// TIA Portal project "TronCamTuDong" (V16)

(* hardware
DEVICE "S7-1200 station_1"  S7-1200 Station
   slot 0: "Rack_0"  S7-1200 Rack  Rack  V1.0
   slot 1: "PLC_1"  CPU 1214C AC/DC/Rly  6ES7 214-1BG40-0XB0  V4.2
*)

// ===== PLC "PLC_1"  CPU 1214C AC/DC/Rly =====

VAR_GLOBAL   // PLC tag table "Input"
   "I_Start" AT %I0.0 : Bool;   // Nút nhấn Start
   "I_Stop" AT %I0.1 : Bool;   // Nút nhấn Stop
   "I_Mode" AT %I0.2 : Bool;   // Công tắc chọn chế độ vận hành
   "I_Ss_Low_XiloA1" AT %I0.3 : Bool;   // Cảm biến xi lô A1
   "I_Ss_Low_XiloA2" AT %I0.4 : Bool;   // Cảm biến xi lô A2
   "I_Ss_Low_XiloA3" AT %I0.5 : Bool;   // Cảm biến xi lô A3
   "I_Ss_Low_XiloA4" AT %I0.6 : Bool;   // Cảm biến xi lô A4
   "I_Ss_Low_XiloA5" AT %I0.7 : Bool;   // Cảm biến xi lô A5
   "I_Ss_Low_XiloA6" AT %I1.0 : Bool;   // Cảm biến xi lô A6
   "I_Ss_Low_XiloA7" AT %I1.1 : Bool;   // Cảm biến xi lô A7
   "I_Ss_Low_XiloA8" AT %I1.2 : Bool;   // Cảm biến xi lô A8
   "I_Ss_Low_XiloA9" AT %I1.3 : Bool;   // Cảm biến xi lô A9
   "I_Ss_Low_XiloB1" AT %I1.4 : Bool;   // Cảm biến xi lô B1
   "I_Ss_Low_XiloB2" AT %I1.5 : Bool;   // Cảm biến xi lô B2
   "I_Ss_Low_XiloB3" AT %I1.6 : Bool;   // Cảm biến xi lô B3
   "I_Ss_Low_XiloB4" AT %I1.7 : Bool;   // Cảm biến xi lô B4
   "I_Ss_Low_XiloB5" AT %I2.0 : Bool;   // Cảm biến xi lô B5
   "I_Ss_Low_XiloB6" AT %I2.1 : Bool;   // Cảm biến xi lô B6
   "I_Ss_Low_XiloB7" AT %I2.2 : Bool;   // Cảm biến xi lô B7
   "I_Ss_ValvesA" AT %I2.3 : Bool;   // Cảm biến van ở thùng cân A
   "I_Ss_ValvesB" AT %I2.4 : Bool;   // Cảm biến van ở thùng cân B
   "I_Ss_Tank_Low" AT %I2.5 : Bool;   // Cảm biến mức thấp bình trộn
   "I_Ss_Tank_High" AT %I2.6 : Bool;   // Cảm biến mức cao bình trộn
   "I_Ss_Valves_Out" AT %I2.7 : Bool;   // Cảm biến van xả ở bình trộn
   "I_SW_Motor_Tai" AT %I3.0 : Bool;   // Công tắc chế độ thủ công động cơ vít tải
   "I_SW_Motor_Mixed" AT %I3.1 : Bool;   // Công tắc chế độ thủ công động cơ trộn
   "I_SW_ValvesA" AT %I3.2 : Bool;   // Công tắc chế độ thủ công van xả thùng cân A
   "I_SW_ValvesB" AT %I3.3 : Bool;   // Công tắc chế độ thủ công van xả thùng cân B
   "I_SW_Valves_Out" AT %I3.4 : Bool;   // Công tắc chế độ thủ công van xả bình trộn
   "I_Load_ScalesA" AT %ID4 : Real;   // Cảm biến cân thùng cân A
   "I_Load_ScalesB" AT %ID8 : Real;   // Cảm biến cân thùng cân B
END_VAR

VAR_GLOBAL   // PLC tag table "Output"
   "Q_lamp_Auto" AT %Q0.0 : Bool;   // Đèn báo chế độ tự động
   "Q_lamp_Manu" AT %Q0.1 : Bool;   // Đèn báo chế độ thủ công
   "Q_lamp_Fault" AT %Q0.2 : Bool;   // Đèn báo lỗi
   "Q_Motor_Tai" AT %Q0.3 : Bool;   // Động cơ vít tải
   "Q_ValveA" AT %Q0.4 : Bool;   // Van xả thùng cân A
   "Q_ValveB" AT %Q0.5 : Bool;   // Van xả thùng cân B
   "Q_Valve_Out" AT %Q0.6 : Bool;   // Van xả bình trộn
   "Q_Motor_Mixed" AT %Q0.7 : Bool;   // Động cơ trộn
   "Q_Motor_Conveyor" AT %Q1.0 : Bool;   // Động cơ điều khiển băng tải
END_VAR

VAR_GLOBAL   // PLC tag table "Output_Auto"
   "M_Auto_Motor_Tai" AT %M20.0 : Bool;
   "M_Auto_ValveA" AT %M20.1 : Bool;
   "M_Auto_ValveB" AT %M20.2 : Bool;
   "M_Auto_Valve_Out" AT %M20.3 : Bool;
   "M_Auto_Motor_Mixed" AT %M20.4 : Bool;
END_VAR

VAR_GLOBAL   // PLC tag table "Output_Manu"
   "M_Manu_Motor_Tai" AT %M30.0 : Bool;
   "M_Manu_ValveA" AT %M30.1 : Bool;
   "M_Manu_ValveB" AT %M30.2 : Bool;
   "M_Manu_Valve_Out" AT %M30.3 : Bool;
   "M_Manu_Motor_Mixed" AT %M30.4 : Bool;
END_VAR

VAR_GLOBAL   // PLC tag table "TrungGian"
   "M_LoadXilo" AT %M15.0 : Bool;
   "M_DK_VanHanh" AT %M15.1 : Bool;
   "M_Step1" AT %M15.2 : Bool;
   "M_Step3" AT %M15.4 : Bool;
   "M_Xung200ms" AT %M15.5 : Bool;
   "M_TG_Laplai" AT %M16.3 : Bool;
   "M_CloseValve1" AT %M16.4 : Bool;
   "M_CloseValve2" AT %M16.5 : Bool;
   "M_Close_MotorTai" AT %M16.6 : Bool;
   "M_Close_MotorMixed" AT %M16.7 : Bool;
   "M_Close_ValveOut" AT %M17.0 : Bool;
   "M_Reset" AT %M17.1 : Bool;
   "M_Step2" AT %M15.3 : Bool;
END_VAR

VAR_GLOBAL   // PLC tag table "TG_Cell_Xilo"
   "M_ScalesA" AT %MD120 : Real;
   "M_ScalesB" AT %MD124 : Real;
   "M_Inverter" AT %MD148 : Real;
END_VAR

DATA_BLOCK "Input"   // DB1
{ S7_Optimized_Access := 'FALSE' }
VERSION : 0.1
   VAR
      Start : Bool;
      Stop : Bool;
      Mode : Bool;
      Simulation : Bool;
      Ss_Low_XiloA1 : Bool;
      Ss_Low_XiloA2 : Bool;
      Ss_Low_XiloA3 : Bool;
      Ss_Low_XiloA4 : Bool;
      Ss_Low_XiloA5 : Bool;
      Ss_Low_XiloA6 : Bool;
      Ss_Low_XiloA7 : Bool;
      Ss_Low_XiloA8 : Bool;
      Ss_Low_XiloA9 : Bool;
      Ss_Low_XiloB1 : Bool;
      Ss_Low_XiloB2 : Bool;
      Ss_Low_XiloB3 : Bool;
      Ss_Low_XiloB4 : Bool;
      Ss_Low_XiloB5 : Bool;
      Ss_Low_XiloB6 : Bool;
      Ss_Low_XiloB7 : Bool;
      Ss_ScalesA : Bool;
      Ss_ScalesB : Bool;
      Ss_Tank_Low : Bool;
      Ss_Tank_High : Bool;
      Ss_Valves_Out : Bool;
      SW_Motor_Tai : Bool;
      SW_Motor_Mixed : Bool;
      SW_ValvesA : Bool;
      SW_ValvesB : Bool;
      SW_Valves_Out : Bool;
   END_VAR
BEGIN
END_DATA_BLOCK

DATA_BLOCK "Output"   // DB2
{ S7_Optimized_Access := 'FALSE' }
VERSION : 0.1
   VAR
      Lamp_Auto : Bool;
      Lamp_Manu : Bool;
      Lamp_Fault : Bool;
      Motor_Tai : Bool;
      ValveA : Bool;
      ValveB : Bool;
      Valve_Out : Bool;
      Motor_Mixed : Bool;
      EndSystem : Bool;
      Act_SoMeTron : Int;
      Act_Weight_XiloA1 : Real;
      Act_Weight_XiloA2 : Real;
      Act_Weight_XiloA3 : Real;
      Act_Weight_XiloA4 : Real;
      Act_Weight_XiloA5 : Real;
      Act_Weight_XiloA6 : Real;
      Act_Weight_XiloA7 : Real;
      Act_Weight_XiloA8 : Real;
      Act_Weight_XiloA9 : Real;
      Act_Weight_XiloB1 : Real;
      Act_Weight_XiloB2 : Real;
      Act_Weight_XiloB3 : Real;
      Act_Weight_XiloB4 : Real;
      Act_Weight_XiloB5 : Real;
      Act_Weight_XiloB6 : Real;
      Act_Weight_XiloB7 : Real;
      Act_Time_Xa : DInt;
      Act_Time_Tron : DInt;
   END_VAR
BEGIN
END_DATA_BLOCK

DATA_BLOCK "Input_Data"   // DB10
{ S7_Optimized_Access := 'FALSE' }
VERSION : 0.1
   VAR
      Load_ScaleA : Real;
      Load_ScaleB : Real;
      Set_Weight_Gao : Real;
      Set_Weight_Ngo : Real;
      Set_Weight_San : Real;
      Set_Weight_DauKho : Real;
      Set_Weight_BotCa : Real;
      Set_Time_Xa : DInt;
      Set_Time_Tron : DInt;
      Set_SoMeTron : Int;
   END_VAR
BEGIN
END_DATA_BLOCK

DATA_BLOCK "DB_TrungGian"   // DB11
{ S7_Optimized_Access := 'FALSE' }
VERSION : 0.1
   VAR
      Enable_XiloGao : Bool;
      Enable_XiloNgo : Bool;
      Enable_XiloSan : Bool;
      Enable_XiloDauKho : Bool;
      Enable_XiloBotca : Bool;
      Xung_200ms : Bool;
   END_VAR
BEGIN
END_DATA_BLOCK

// folder: System blocks/Program resources

DATA_BLOCK "Xung200ms"   // DB3
{ S7_Optimized_Access := 'TRUE' }
AUTHOR : Simatic
FAMILY : IEC
NAME : IEC_TMR
VERSION : 1.0
// stored: InstanceOfName IEC_TIMER
"IEC_TIMER"
BEGIN
END_DATA_BLOCK

DATA_BLOCK "Time_Mix"   // DB4
{ S7_Optimized_Access := 'TRUE' }
AUTHOR : Simatic
FAMILY : IEC
NAME : IEC_TMR
VERSION : 1.0
// stored: InstanceOfName IEC_TIMER
"IEC_TIMER"
BEGIN
END_DATA_BLOCK

DATA_BLOCK "Time_Xa"   // DB5
{ S7_Optimized_Access := 'TRUE' }
AUTHOR : Simatic
FAMILY : IEC
NAME : IEC_TMR
VERSION : 1.0
// stored: InstanceOfName IEC_TIMER
"IEC_TIMER"
BEGIN
END_DATA_BLOCK

DATA_BLOCK "TimeDelay"   // DB6
{ S7_Optimized_Access := 'TRUE' }
AUTHOR : Simatic
FAMILY : IEC
NAME : IEC_TMR
VERSION : 1.0
// stored: InstanceOfName IEC_TIMER
"IEC_TIMER"
BEGIN
END_DATA_BLOCK

DATA_BLOCK "TimeDelay2"   // DB7
{ S7_Optimized_Access := 'TRUE' }
AUTHOR : Simatic
FAMILY : IEC
NAME : IEC_TMR
VERSION : 1.0
// stored: InstanceOfName IEC_TIMER
"IEC_TIMER"
BEGIN
END_DATA_BLOCK

DATA_BLOCK "Dem_SoMe"   // DB8
{ S7_Optimized_Access := 'TRUE' }
AUTHOR : Simatic
FAMILY : IEC
NAME : CNTR
VERSION : 1.0
// stored: InstanceOfName IEC_COUNTER
"IEC_COUNTER"
BEGIN
END_DATA_BLOCK

DATA_BLOCK "Time_Delay3"   // DB9
{ S7_Optimized_Access := 'TRUE' }
AUTHOR : Simatic
FAMILY : IEC
NAME : IEC_TMR
VERSION : 1.0
// stored: InstanceOfName IEC_TIMER
"IEC_TIMER"
BEGIN
END_DATA_BLOCK

// folder: (top level)

FUNCTION "FC_Auto" : Void   // FC1, LAD
{ S7_Optimized_Access := 'TRUE' }
VERSION : 0.1
   VAR_TEMP   // added for the SCL form of the ladder/FBD networks
      _w1 : Bool;
   END_VAR
BEGIN

REGION Network 1: kiểm tra điều kiện các giá trị khối lượng n.liệu và t.gian xả , trộn > 0
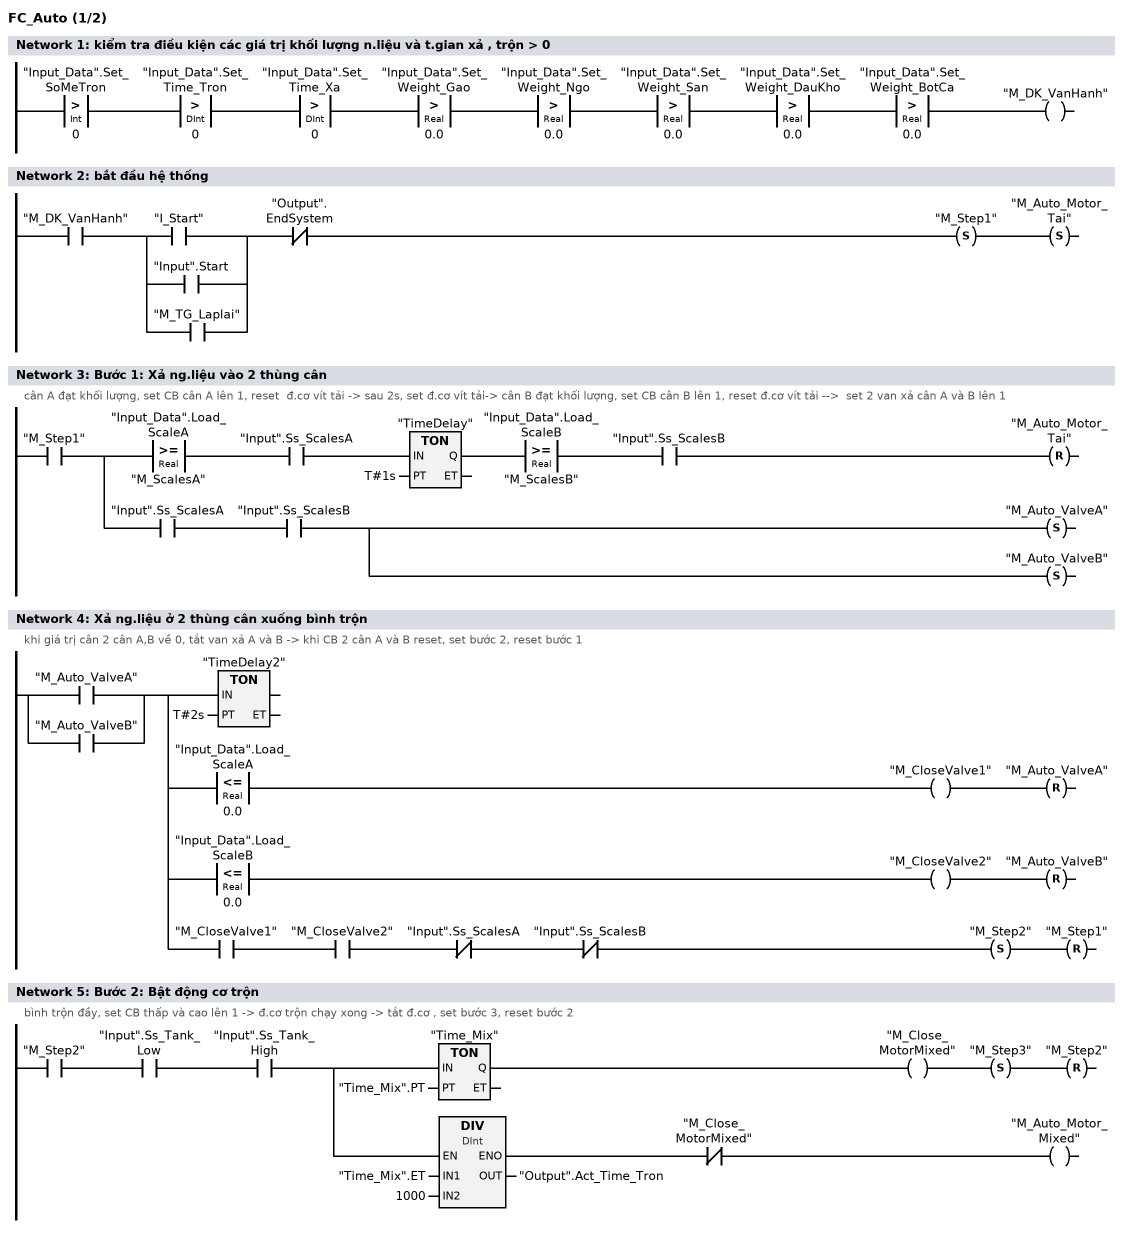
   RUNG wire#powerrail
      { S7_Templates := "SrcType := Int" } GT_Contact(in1 := "Input_Data".Set_SoMeTron, in2 := 0)
      { S7_Templates := "SrcType := DInt" } GT_Contact(in1 := "Input_Data".Set_Time_Tron, in2 := 0)
      { S7_Templates := "SrcType := DInt" } GT_Contact(in1 := "Input_Data".Set_Time_Xa, in2 := 0)
      { S7_Templates := "SrcType := Real" } GT_Contact(in1 := "Input_Data".Set_Weight_Gao, in2 := 0.0)
      { S7_Templates := "SrcType := Real" } GT_Contact(in1 := "Input_Data".Set_Weight_Ngo, in2 := 0.0)
      { S7_Templates := "SrcType := Real" } GT_Contact(in1 := "Input_Data".Set_Weight_San, in2 := 0.0)
      { S7_Templates := "SrcType := Real" } GT_Contact(in1 := "Input_Data".Set_Weight_DauKho, in2 := 0.0)
      { S7_Templates := "SrcType := Real" } GT_Contact(in1 := "Input_Data".Set_Weight_BotCa, in2 := 0.0)
      Coil( "M_DK_VanHanh" )
   END_RUNG
   // the same network as SCL:
   "M_DK_VanHanh" := ("Input_Data".Set_SoMeTron > 0) AND ("Input_Data".Set_Time_Tron > 0) AND ("Input_Data".Set_Time_Xa > 0) AND ("Input_Data".Set_Weight_Gao > 0.0) AND ("Input_Data".Set_Weight_Ngo > 0.0) AND ("Input_Data".Set_Weight_San > 0.0) AND ("Input_Data".Set_Weight_DauKho > 0.0) AND ("Input_Data".Set_Weight_BotCa > 0.0);
END_REGION

REGION Network 2: bắt đầu hệ thống
   RUNG wire#powerrail
      Contact( "M_DK_VanHanh" )
      wire#w1
      Contact( "I_Start" )
      wire#w2
      I_Contact( "Output".EndSystem )
      S_Coil( "M_Step1" )
      S_Coil( "M_Auto_Motor_Tai" )
   END_RUNG
   RUNG wire#w1
      Contact( "Input".Start )
   END_RUNG wire#w2
   RUNG wire#w1
      Contact( "M_TG_Laplai" )
   END_RUNG wire#w2
   // the same network as SCL:
   IF "M_DK_VanHanh" AND ("I_Start" OR "Input".Start OR "M_TG_Laplai") AND NOT "Output".EndSystem THEN
       "M_Step1" := TRUE;
       "M_Auto_Motor_Tai" := TRUE;
   END_IF;
END_REGION

REGION Network 3: Bước 1: Xả ng.liệu vào 2 thùng cân
   // cân A đạt khối lượng, set CB cân A lên 1, reset  đ.cơ vít tải -> sau 2s, set đ.cơ vít tải-> cân B đạt khối lượng, set CB cân B lên 1, reset đ.cơ vít tải -->  set 2 van xả cân A và B lên 1
   "TimeDelay".TON(IN := "M_Step1" AND ("Input_Data".Load_ScaleA >= "M_ScalesA") AND "Input".Ss_ScalesA,
                   PT := T#1s);
   IF "TimeDelay".Q AND ("Input_Data".Load_ScaleB >= "M_ScalesB") AND "Input".Ss_ScalesB THEN
       "M_Auto_Motor_Tai" := FALSE;
   END_IF;
   IF "M_Step1" AND "Input".Ss_ScalesA AND "Input".Ss_ScalesB THEN
       "M_Auto_ValveA" := TRUE;
       "M_Auto_ValveB" := TRUE;
   END_IF;
END_REGION

REGION Network 4: Xả ng.liệu ở 2 thùng cân xuống bình trộn
   // khi giá trị cân 2 cân A,B về 0, tắt van xả A và B -> khi CB 2 cân A và B reset, set bước 2, reset bước 1
   #_w1 := "M_Auto_ValveA" OR "M_Auto_ValveB";
   "TimeDelay2".TON(IN := #_w1, PT := T#2s);
   "M_CloseValve1" := #_w1 AND ("Input_Data".Load_ScaleA <= 0.0);
   IF "M_CloseValve1" THEN "M_Auto_ValveA" := FALSE; END_IF;
   "M_CloseValve2" := #_w1 AND ("Input_Data".Load_ScaleB <= 0.0);
   IF "M_CloseValve2" THEN "M_Auto_ValveB" := FALSE; END_IF;
   IF #_w1 AND "M_CloseValve1" AND "M_CloseValve2" AND NOT "Input".Ss_ScalesA AND NOT "Input".Ss_ScalesB THEN
       "M_Step2" := TRUE;
       "M_Step1" := FALSE;
   END_IF;
END_REGION

REGION Network 5: Bước 2: Bật động cơ trộn
   // bình trộn đầy, set CB thấp và cao lên 1 -> đ.cơ trộn chạy xong -> tắt đ.cơ , set bước 3, reset bước 2
   #_w1 := "M_Step2" AND "Input".Ss_Tank_Low AND "Input".Ss_Tank_High;
   "Time_Mix".TON(IN := #_w1, PT := "Time_Mix".PT);
   "M_Close_MotorMixed" := "Time_Mix".Q;
   IF "Time_Mix".Q THEN
       "M_Step3" := TRUE;
       "M_Step2" := FALSE;
   END_IF;
   IF #_w1 THEN "Output".Act_Time_Tron := "Time_Mix".ET / 1000; END_IF;
   "M_Auto_Motor_Mixed" := #_w1 AND NOT "M_Close_MotorMixed";
END_REGION

REGION Network 6: Bước 3: bật van xả liệu đầu ra
   // CB cao bình trộn reset , bắt đầu xả -> xả xong , CB thấp reset , tắt van xả đầu ra --> set biến lặp lại, reset bước 3
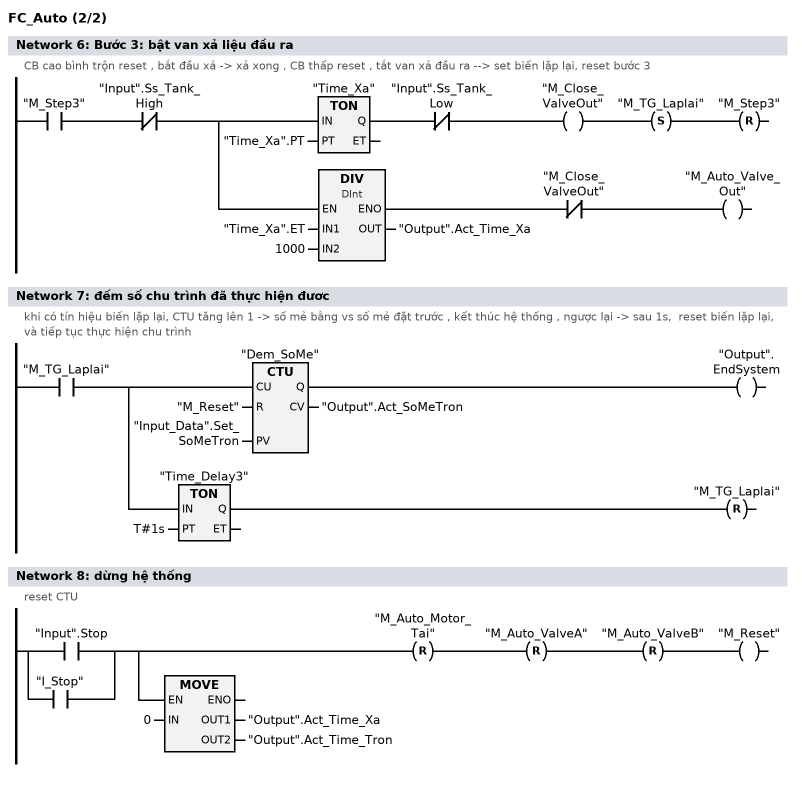
   #_w1 := "M_Step3" AND NOT "Input".Ss_Tank_High;
   "Time_Xa".TON(IN := #_w1, PT := "Time_Xa".PT);
   "M_Close_ValveOut" := "Time_Xa".Q AND NOT "Input".Ss_Tank_Low;
   IF "M_Close_ValveOut" THEN
       "M_TG_Laplai" := TRUE;
       "M_Step3" := FALSE;
   END_IF;
   IF #_w1 THEN "Output".Act_Time_Xa := "Time_Xa".ET / 1000; END_IF;
   "M_Auto_Valve_Out" := #_w1 AND NOT "M_Close_ValveOut";
END_REGION

REGION Network 7: đếm số chu trình đã thực hiện đươc
   // khi có tín hiệu biến lặp lại, CTU tăng lên 1 -> số mẻ bằng vs số mẻ đặt trước , kết thúc hệ thống , ngược lại -> sau 1s,  reset biến lặp lại, và tiếp tục thực hiện chu trình
   "Dem_SoMe".CTU(CU := "M_TG_Laplai",
                  R := "M_Reset",
                  PV := "Input_Data".Set_SoMeTron,
                  CV => "Output".Act_SoMeTron);
   "Output".EndSystem := "Dem_SoMe".Q;
   "Time_Delay3".TON(IN := "M_TG_Laplai", PT := T#1s);
   IF "Time_Delay3".Q THEN "M_TG_Laplai" := FALSE; END_IF;
END_REGION

REGION Network 8: dừng hệ thống
   // reset CTU
   RUNG wire#powerrail
      Contact( "Input".Stop )
      wire#w1
      R_Coil( "M_Auto_Motor_Tai" )
      R_Coil( "M_Auto_ValveA" )
      R_Coil( "M_Auto_ValveB" )
      Coil( "M_Reset" )
   END_RUNG
   RUNG wire#powerrail
      Contact( "I_Stop" )
   END_RUNG wire#w1
   RUNG wire#w1
      Move(in := 0, out1 => "Output".Act_Time_Xa, out2 => "Output".Act_Time_Tron)
   END_RUNG
   // the same network as SCL:
   #_w1 := "Input".Stop OR "I_Stop";
   IF #_w1 THEN
       "M_Auto_Motor_Tai" := FALSE;
       "M_Auto_ValveA" := FALSE;
       "M_Auto_ValveB" := FALSE;
   END_IF;
   "M_Reset" := #_w1;
   IF #_w1 THEN
       "Output".Act_Time_Xa := 0;
       "Output".Act_Time_Tron := 0;
   END_IF;
END_REGION
END_FUNCTION

FUNCTION "FC_Manu" : Void   // FC2, LAD
{ S7_Optimized_Access := 'TRUE' }
VERSION : 0.1
BEGIN

REGION Network 1: bật/ tắt đ.cơ tải
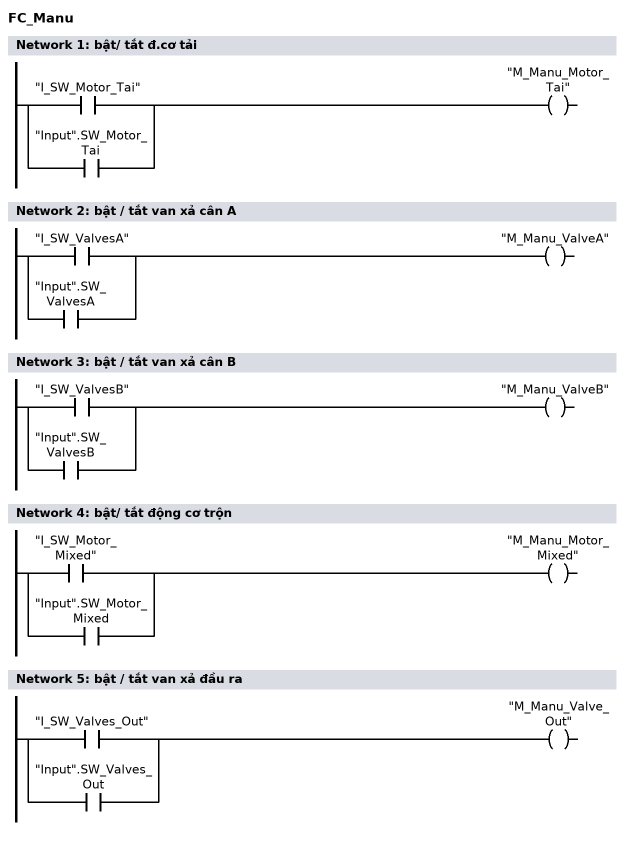
   RUNG wire#powerrail
      Contact( "I_SW_Motor_Tai" )
      wire#w1
      Coil( "M_Manu_Motor_Tai" )
   END_RUNG
   RUNG wire#powerrail
      Contact( "Input".SW_Motor_Tai )
   END_RUNG wire#w1
   // the same network as SCL:
   "M_Manu_Motor_Tai" := "I_SW_Motor_Tai" OR "Input".SW_Motor_Tai;
END_REGION

REGION Network 2: bật / tắt van xả cân A
   RUNG wire#powerrail
      Contact( "I_SW_ValvesA" )
      wire#w1
      Coil( "M_Manu_ValveA" )
   END_RUNG
   RUNG wire#powerrail
      Contact( "Input".SW_ValvesA )
   END_RUNG wire#w1
   // the same network as SCL:
   "M_Manu_ValveA" := "I_SW_ValvesA" OR "Input".SW_ValvesA;
END_REGION

REGION Network 3: bật / tắt van xả cân B
   RUNG wire#powerrail
      Contact( "I_SW_ValvesB" )
      wire#w1
      Coil( "M_Manu_ValveB" )
   END_RUNG
   RUNG wire#powerrail
      Contact( "Input".SW_ValvesB )
   END_RUNG wire#w1
   // the same network as SCL:
   "M_Manu_ValveB" := "I_SW_ValvesB" OR "Input".SW_ValvesB;
END_REGION

REGION Network 4: bật/ tắt động cơ trộn
   RUNG wire#powerrail
      Contact( "I_SW_Motor_Mixed" )
      wire#w1
      Coil( "M_Manu_Motor_Mixed" )
   END_RUNG
   RUNG wire#powerrail
      Contact( "Input".SW_Motor_Mixed )
   END_RUNG wire#w1
   // the same network as SCL:
   "M_Manu_Motor_Mixed" := "I_SW_Motor_Mixed" OR "Input".SW_Motor_Mixed;
END_REGION

REGION Network 5: bật / tắt van xả đầu ra
   RUNG wire#powerrail
      Contact( "I_SW_Valves_Out" )
      wire#w1
      Coil( "M_Manu_Valve_Out" )
   END_RUNG
   RUNG wire#powerrail
      Contact( "Input".SW_Valves_Out )
   END_RUNG wire#w1
   // the same network as SCL:
   "M_Manu_Valve_Out" := "I_SW_Valves_Out" OR "Input".SW_Valves_Out;
END_REGION
END_FUNCTION

FUNCTION "FC_Simulation" : Void   // FC3, LAD
{ S7_Optimized_Access := 'TRUE' }
VERSION : 0.1
   VAR_TEMP   // added for the SCL form of the ladder/FBD networks
      _w1 : Bool;
      _w2 : Bool;
      _w3 : Bool;
      _w4 : Bool;
   END_VAR
BEGIN

REGION Network 1: tạo xung 200ms
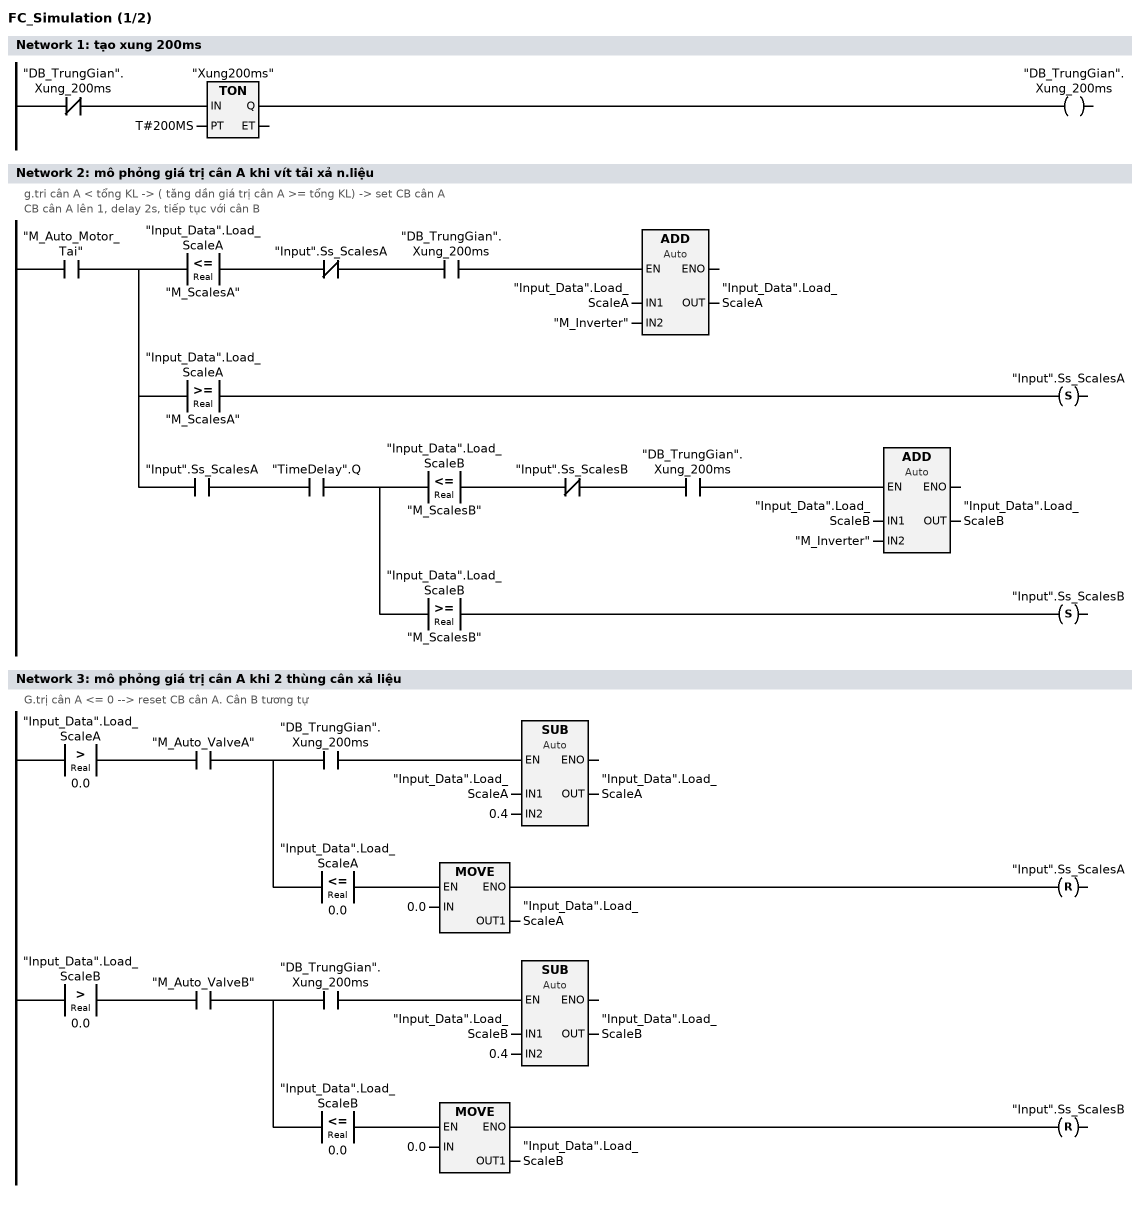
   "Xung200ms".TON(IN := NOT "DB_TrungGian".Xung_200ms, PT := T#200MS);
   "DB_TrungGian".Xung_200ms := "Xung200ms".Q;
END_REGION

REGION Network 2: mô phỏng giá trị cân A khi vít tải xả n.liệu
   // g.tri cân A < tổng KL -> ( tăng dần giá trị cân A >= tổng KL) -> set CB cân A 
   // CB cân A lên 1, delay 2s, tiếp tục với cân B
   RUNG wire#powerrail
      Contact( "M_Auto_Motor_Tai" )
      wire#w1
      { S7_Templates := "SrcType := Real" } LE_Contact(in1 := "Input_Data".Load_ScaleA, in2 := "M_ScalesA")
      I_Contact( "Input".Ss_ScalesA )
      Contact( "DB_TrungGian".Xung_200ms )
      Add(in1 := "Input_Data".Load_ScaleA, in2 := "M_Inverter", out => "Input_Data".Load_ScaleA)
   END_RUNG
   RUNG wire#w1
      { S7_Templates := "SrcType := Real" } GE_Contact(in1 := "Input_Data".Load_ScaleA, in2 := "M_ScalesA")
      S_Coil( "Input".Ss_ScalesA )
   END_RUNG
   RUNG wire#w1
      Contact( "Input".Ss_ScalesA )
      Contact( "TimeDelay".Q )
      wire#w2
      { S7_Templates := "SrcType := Real" } LE_Contact(in1 := "Input_Data".Load_ScaleB, in2 := "M_ScalesB")
      I_Contact( "Input".Ss_ScalesB )
      Contact( "DB_TrungGian".Xung_200ms )
      Add(in1 := "Input_Data".Load_ScaleB, in2 := "M_Inverter", out => "Input_Data".Load_ScaleB)
   END_RUNG
   RUNG wire#w2
      { S7_Templates := "SrcType := Real" } GE_Contact(in1 := "Input_Data".Load_ScaleB, in2 := "M_ScalesB")
      S_Coil( "Input".Ss_ScalesB )
   END_RUNG
   // the same network as SCL:
   IF "M_Auto_Motor_Tai" AND ("Input_Data".Load_ScaleA <= "M_ScalesA") AND NOT "Input".Ss_ScalesA AND "DB_TrungGian".Xung_200ms THEN
       "Input_Data".Load_ScaleA := "Input_Data".Load_ScaleA + "M_Inverter";
   END_IF;
   IF "M_Auto_Motor_Tai" AND ("Input_Data".Load_ScaleA >= "M_ScalesA") THEN
       "Input".Ss_ScalesA := TRUE;
   END_IF;
   #_w1 := "M_Auto_Motor_Tai" AND "Input".Ss_ScalesA AND "TimeDelay".Q;
   IF #_w1 AND ("Input_Data".Load_ScaleB <= "M_ScalesB") AND NOT "Input".Ss_ScalesB AND "DB_TrungGian".Xung_200ms THEN
       "Input_Data".Load_ScaleB := "Input_Data".Load_ScaleB + "M_Inverter";
   END_IF;
   IF #_w1 AND ("Input_Data".Load_ScaleB >= "M_ScalesB") THEN "Input".Ss_ScalesB := TRUE; END_IF;
END_REGION

REGION Network 3: mô phỏng giá trị cân A khi 2 thùng cân xả liệu
   // G.trị cân A <= 0 --> reset CB cân A. Cân B tương tự
   RUNG wire#powerrail
      { S7_Templates := "SrcType := Real" } GT_Contact(in1 := "Input_Data".Load_ScaleA, in2 := 0.0)
      Contact( "M_Auto_ValveA" )
      wire#w1
      Contact( "DB_TrungGian".Xung_200ms )
      Sub(in1 := "Input_Data".Load_ScaleA, in2 := 0.4, out => "Input_Data".Load_ScaleA)
   END_RUNG
   RUNG wire#w1
      { S7_Templates := "SrcType := Real" } LE_Contact(in1 := "Input_Data".Load_ScaleA, in2 := 0.0)
      Move(in := 0.0, out1 => "Input_Data".Load_ScaleA)
      R_Coil( "Input".Ss_ScalesA )
   END_RUNG
   RUNG wire#powerrail
      { S7_Templates := "SrcType := Real" } GT_Contact(in1 := "Input_Data".Load_ScaleB, in2 := 0.0)
      Contact( "M_Auto_ValveB" )
      wire#w2
      Contact( "DB_TrungGian".Xung_200ms )
      Sub(in1 := "Input_Data".Load_ScaleB, in2 := 0.4, out => "Input_Data".Load_ScaleB)
   END_RUNG
   RUNG wire#w2
      { S7_Templates := "SrcType := Real" } LE_Contact(in1 := "Input_Data".Load_ScaleB, in2 := 0.0)
      Move(in := 0.0, out1 => "Input_Data".Load_ScaleB)
      R_Coil( "Input".Ss_ScalesB )
   END_RUNG
   // the same network as SCL:
   #_w1 := ("Input_Data".Load_ScaleA > 0.0) AND "M_Auto_ValveA";
   IF #_w1 AND "DB_TrungGian".Xung_200ms THEN
       "Input_Data".Load_ScaleA := "Input_Data".Load_ScaleA - 0.4;
   END_IF;
   #_w2 := #_w1 AND ("Input_Data".Load_ScaleA <= 0.0);
   IF #_w2 THEN
       "Input_Data".Load_ScaleA := 0.0;
       "Input".Ss_ScalesA := FALSE;
   END_IF;
   #_w3 := ("Input_Data".Load_ScaleB > 0.0) AND "M_Auto_ValveB";
   IF #_w3 AND "DB_TrungGian".Xung_200ms THEN
       "Input_Data".Load_ScaleB := "Input_Data".Load_ScaleB - 0.4;
   END_IF;
   #_w4 := #_w3 AND ("Input_Data".Load_ScaleB <= 0.0);
   IF #_w4 THEN
       "Input_Data".Load_ScaleB := 0.0;
       "Input".Ss_ScalesB := FALSE;
   END_IF;
END_REGION

REGION Network 4
   // Khi 2 thùng cân bắt đầu xả , sau 2s , set CB thấp. Sau khi xả hết 2 thùng, set bước 2 và set CB cao
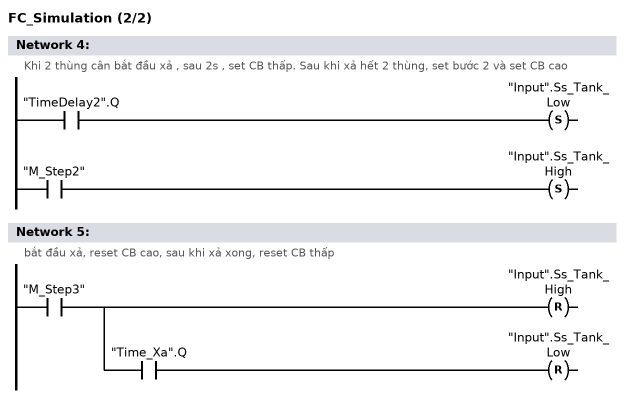
   RUNG wire#powerrail
      Contact( "TimeDelay2".Q )
      S_Coil( "Input".Ss_Tank_Low )
   END_RUNG
   RUNG wire#powerrail
      Contact( "M_Step2" )
      S_Coil( "Input".Ss_Tank_High )
   END_RUNG
   // the same network as SCL:
   IF "TimeDelay2".Q THEN "Input".Ss_Tank_Low := TRUE; END_IF;
   IF "M_Step2" THEN "Input".Ss_Tank_High := TRUE; END_IF;
END_REGION

REGION Network 5
   // bắt đầu xả, reset CB cao, sau khi xả xong, reset CB thấp
   RUNG wire#powerrail
      Contact( "M_Step3" )
      wire#w1
      R_Coil( "Input".Ss_Tank_High )
   END_RUNG
   RUNG wire#w1
      Contact( "Time_Xa".Q )
      R_Coil( "Input".Ss_Tank_Low )
   END_RUNG
   // the same network as SCL:
   IF "M_Step3" THEN "Input".Ss_Tank_High := FALSE; END_IF;
   IF "M_Step3" AND "Time_Xa".Q THEN "Input".Ss_Tank_Low := FALSE; END_IF;
END_REGION
END_FUNCTION

FUNCTION "FC_Output" : Void   // FC4, LAD
{ S7_Optimized_Access := 'TRUE' }
VERSION : 0.1
// set tín hiệu ngõ ra nếu có tín hiệu từ output manu hoặc auto, ngược lại reset tin hiệu
BEGIN

REGION Network 1
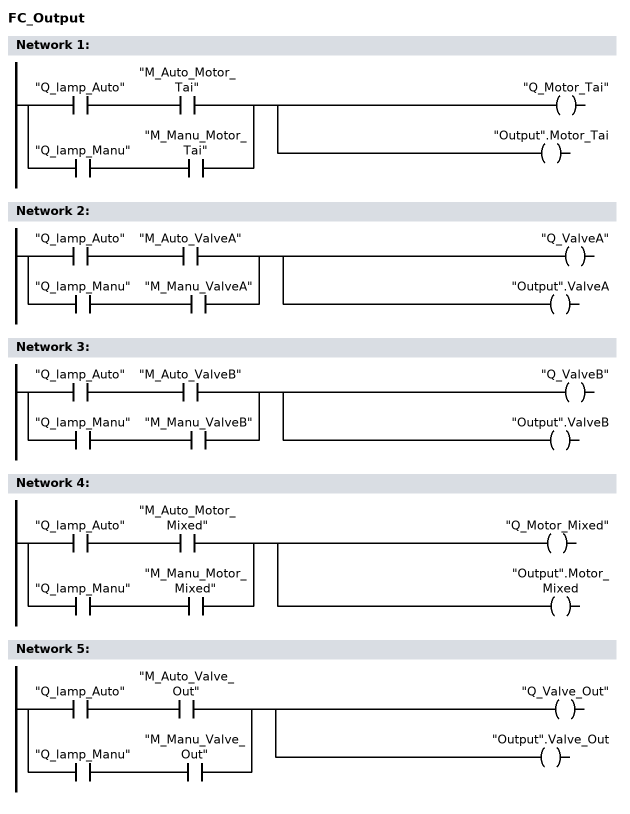
   RUNG wire#powerrail
      Contact( "Q_lamp_Auto" )
      Contact( "M_Auto_Motor_Tai" )
      wire#w1
      Coil( "Q_Motor_Tai" )
   END_RUNG
   RUNG wire#powerrail
      Contact( "Q_lamp_Manu" )
      Contact( "M_Manu_Motor_Tai" )
   END_RUNG wire#w1
   RUNG wire#w1
      Coil( "Output".Motor_Tai )
   END_RUNG
   // the same network as SCL:
   "Q_Motor_Tai" := ("Q_lamp_Auto" AND "M_Auto_Motor_Tai") OR ("Q_lamp_Manu" AND "M_Manu_Motor_Tai");
   "Output".Motor_Tai := "Q_Motor_Tai";
END_REGION

REGION Network 2
   RUNG wire#powerrail
      Contact( "Q_lamp_Auto" )
      Contact( "M_Auto_ValveA" )
      wire#w1
      Coil( "Q_ValveA" )
   END_RUNG
   RUNG wire#powerrail
      Contact( "Q_lamp_Manu" )
      Contact( "M_Manu_ValveA" )
   END_RUNG wire#w1
   RUNG wire#w1
      Coil( "Output".ValveA )
   END_RUNG
   // the same network as SCL:
   "Q_ValveA" := ("Q_lamp_Auto" AND "M_Auto_ValveA") OR ("Q_lamp_Manu" AND "M_Manu_ValveA");
   "Output".ValveA := "Q_ValveA";
END_REGION

REGION Network 3
   RUNG wire#powerrail
      Contact( "Q_lamp_Auto" )
      Contact( "M_Auto_ValveB" )
      wire#w1
      Coil( "Q_ValveB" )
   END_RUNG
   RUNG wire#powerrail
      Contact( "Q_lamp_Manu" )
      Contact( "M_Manu_ValveB" )
   END_RUNG wire#w1
   RUNG wire#w1
      Coil( "Output".ValveB )
   END_RUNG
   // the same network as SCL:
   "Q_ValveB" := ("Q_lamp_Auto" AND "M_Auto_ValveB") OR ("Q_lamp_Manu" AND "M_Manu_ValveB");
   "Output".ValveB := "Q_ValveB";
END_REGION

REGION Network 4
   RUNG wire#powerrail
      Contact( "Q_lamp_Auto" )
      Contact( "M_Auto_Motor_Mixed" )
      wire#w1
      Coil( "Q_Motor_Mixed" )
   END_RUNG
   RUNG wire#powerrail
      Contact( "Q_lamp_Manu" )
      Contact( "M_Manu_Motor_Mixed" )
   END_RUNG wire#w1
   RUNG wire#w1
      Coil( "Output".Motor_Mixed )
   END_RUNG
   // the same network as SCL:
   "Q_Motor_Mixed" := ("Q_lamp_Auto" AND "M_Auto_Motor_Mixed") OR ("Q_lamp_Manu" AND "M_Manu_Motor_Mixed");
   "Output".Motor_Mixed := "Q_Motor_Mixed";
END_REGION

REGION Network 5
   RUNG wire#powerrail
      Contact( "Q_lamp_Auto" )
      Contact( "M_Auto_Valve_Out" )
      wire#w1
      Coil( "Q_Valve_Out" )
   END_RUNG
   RUNG wire#powerrail
      Contact( "Q_lamp_Manu" )
      Contact( "M_Manu_Valve_Out" )
   END_RUNG wire#w1
   RUNG wire#w1
      Coil( "Output".Valve_Out )
   END_RUNG
   // the same network as SCL:
   "Q_Valve_Out" := ("Q_lamp_Auto" AND "M_Auto_Valve_Out") OR ("Q_lamp_Manu" AND "M_Manu_Valve_Out");
   "Output".Valve_Out := "Q_Valve_Out";
END_REGION
END_FUNCTION

FUNCTION "FC_Math" : Void   // FC5, LAD
{ S7_Optimized_Access := 'TRUE' }
VERSION : 0.1
   VAR_TEMP
      sumGaoNgo : Real;
      sumGaoSan : Real;
      sumNgoSan : Real;
   END_VAR
   VAR_TEMP   // added for the SCL form of the ladder/FBD networks
      _w1 : Bool;
      _w2 : Bool;
      _w3 : Bool;
      _w4 : Bool;
      _w5 : Bool;
   END_VAR
BEGIN

REGION Network 1: tính tổng 3 n.liệu gạo, ngô, sắn đưa vào giá trị cân A, đậu khô, bột cá đưa vào g.trị cân B
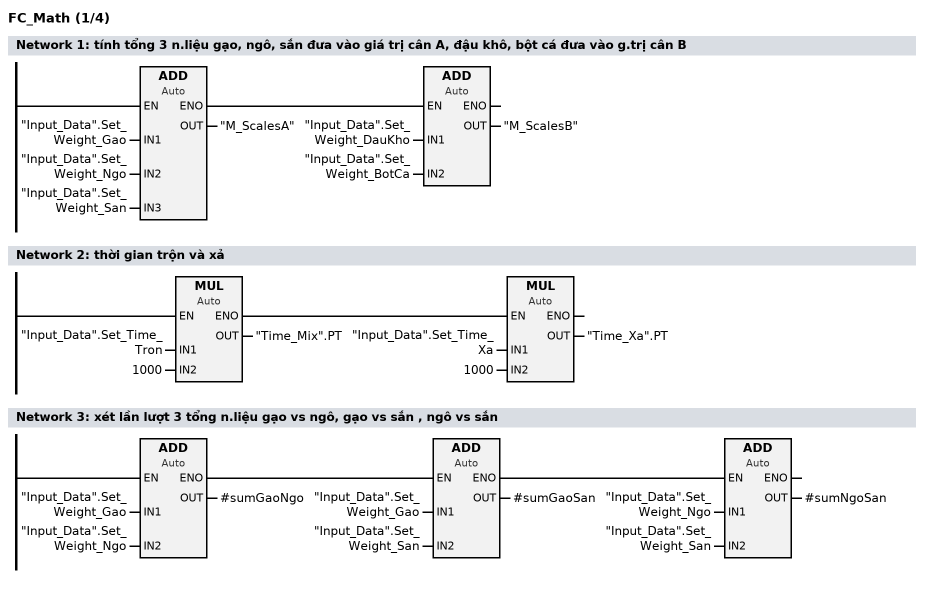
   RUNG wire#powerrail
      Add(in1 := "Input_Data".Set_Weight_Gao, in2 := "Input_Data".Set_Weight_Ngo, in3 := "Input_Data".Set_Weight_San, out => "M_ScalesA")
      Add(in1 := "Input_Data".Set_Weight_DauKho, in2 := "Input_Data".Set_Weight_BotCa, out => "M_ScalesB")
   END_RUNG
   // the same network as SCL:
   "M_ScalesA" := "Input_Data".Set_Weight_Gao + "Input_Data".Set_Weight_Ngo + "Input_Data".Set_Weight_San;
   "M_ScalesB" := "Input_Data".Set_Weight_DauKho + "Input_Data".Set_Weight_BotCa;
END_REGION

REGION Network 2: thời gian trộn và xả
   RUNG wire#powerrail
      Mul(in1 := "Input_Data".Set_Time_Tron, in2 := 1000, out => "Time_Mix".PT)
      Mul(in1 := "Input_Data".Set_Time_Xa, in2 := 1000, out => "Time_Xa".PT)
   END_RUNG
   // the same network as SCL:
   "Time_Mix".PT := "Input_Data".Set_Time_Tron * 1000;
   "Time_Xa".PT := "Input_Data".Set_Time_Xa * 1000;
END_REGION

REGION Network 3: xét lần lượt 3 tổng n.liệu gạo vs ngô, gạo vs sắn , ngô vs sắn
   RUNG wire#powerrail
      Add(in1 := "Input_Data".Set_Weight_Gao, in2 := "Input_Data".Set_Weight_Ngo, out => #sumGaoNgo)
      Add(in1 := "Input_Data".Set_Weight_Gao, in2 := "Input_Data".Set_Weight_San, out => #sumGaoSan)
      Add(in1 := "Input_Data".Set_Weight_Ngo, in2 := "Input_Data".Set_Weight_San, out => #sumNgoSan)
   END_RUNG
   // the same network as SCL:
   #sumGaoNgo := "Input_Data".Set_Weight_Gao + "Input_Data".Set_Weight_Ngo;
   #sumGaoSan := "Input_Data".Set_Weight_Gao + "Input_Data".Set_Weight_San;
   #sumNgoSan := "Input_Data".Set_Weight_Ngo + "Input_Data".Set_Weight_San;
END_REGION

REGION Network 4: so sánh các g.trị nguyên liệu đầu vào của cân A
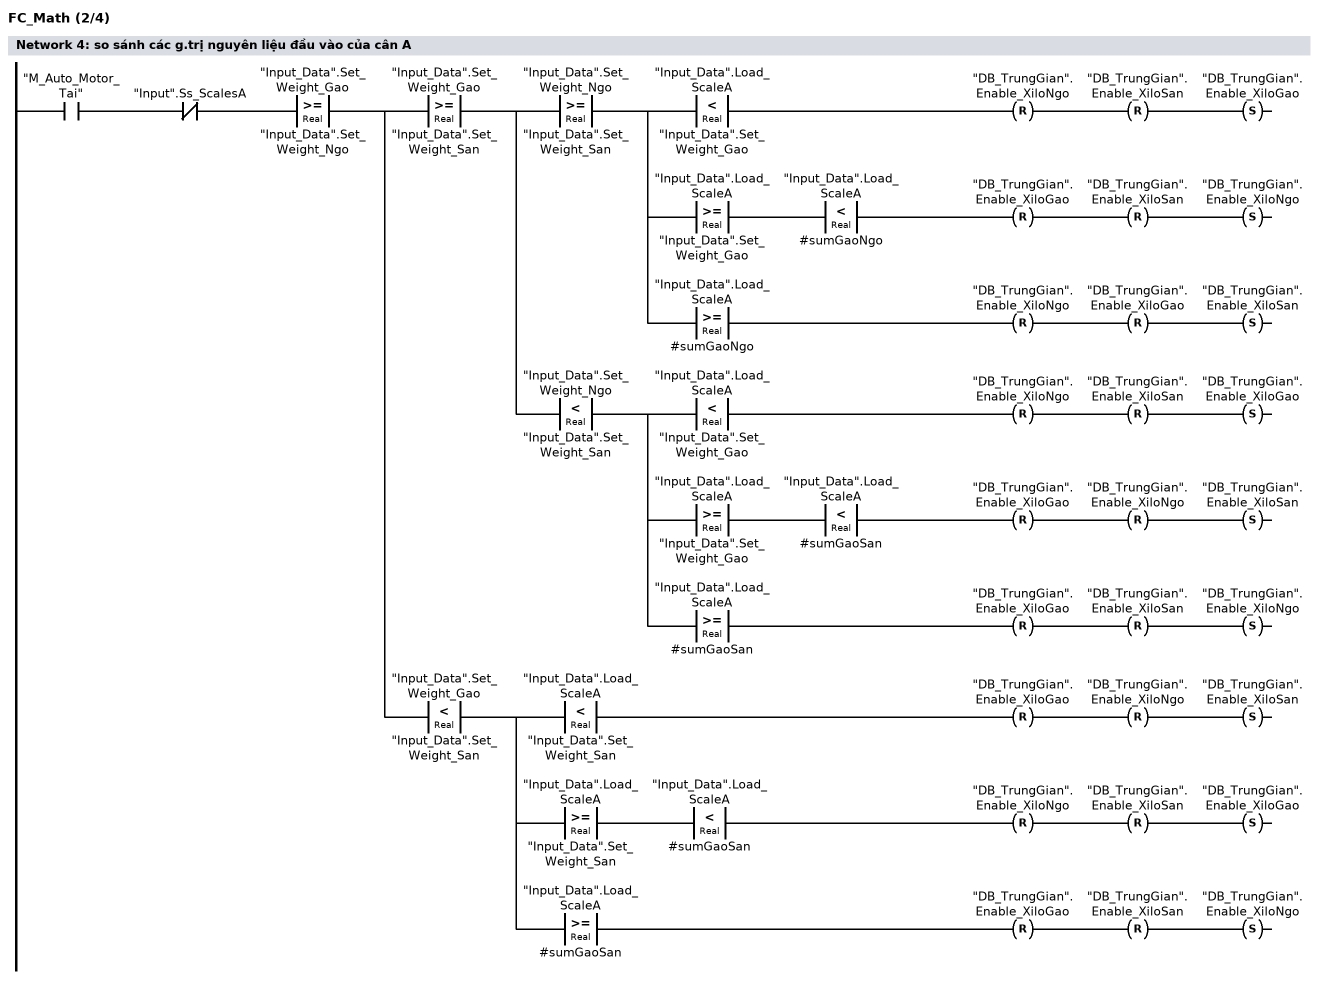
   RUNG wire#powerrail
      Contact( "M_Auto_Motor_Tai" )
      I_Contact( "Input".Ss_ScalesA )
      { S7_Templates := "SrcType := Real" } GE_Contact(in1 := "Input_Data".Set_Weight_Gao, in2 := "Input_Data".Set_Weight_Ngo)
      wire#w1
      { S7_Templates := "SrcType := Real" } GE_Contact(in1 := "Input_Data".Set_Weight_Gao, in2 := "Input_Data".Set_Weight_San)
      wire#w2
      { S7_Templates := "SrcType := Real" } GE_Contact(in1 := "Input_Data".Set_Weight_Ngo, in2 := "Input_Data".Set_Weight_San)
      wire#w3
      { S7_Templates := "SrcType := Real" } LT_Contact(in1 := "Input_Data".Load_ScaleA, in2 := "Input_Data".Set_Weight_Gao)
      R_Coil( "DB_TrungGian".Enable_XiloNgo )
      R_Coil( "DB_TrungGian".Enable_XiloSan )
      S_Coil( "DB_TrungGian".Enable_XiloGao )
   END_RUNG
   RUNG wire#w3
      { S7_Templates := "SrcType := Real" } GE_Contact(in1 := "Input_Data".Load_ScaleA, in2 := "Input_Data".Set_Weight_Gao)
      { S7_Templates := "SrcType := Real" } LT_Contact(in1 := "Input_Data".Load_ScaleA, in2 := #sumGaoNgo)
      R_Coil( "DB_TrungGian".Enable_XiloGao )
      R_Coil( "DB_TrungGian".Enable_XiloSan )
      S_Coil( "DB_TrungGian".Enable_XiloNgo )
   END_RUNG
   RUNG wire#w3
      { S7_Templates := "SrcType := Real" } GE_Contact(in1 := "Input_Data".Load_ScaleA, in2 := #sumGaoNgo)
      R_Coil( "DB_TrungGian".Enable_XiloNgo )
      R_Coil( "DB_TrungGian".Enable_XiloGao )
      S_Coil( "DB_TrungGian".Enable_XiloSan )
   END_RUNG
   RUNG wire#w2
      { S7_Templates := "SrcType := Real" } LT_Contact(in1 := "Input_Data".Set_Weight_Ngo, in2 := "Input_Data".Set_Weight_San)
      wire#w4
      { S7_Templates := "SrcType := Real" } LT_Contact(in1 := "Input_Data".Load_ScaleA, in2 := "Input_Data".Set_Weight_Gao)
      R_Coil( "DB_TrungGian".Enable_XiloNgo )
      R_Coil( "DB_TrungGian".Enable_XiloSan )
      S_Coil( "DB_TrungGian".Enable_XiloGao )
   END_RUNG
   RUNG wire#w4
      { S7_Templates := "SrcType := Real" } GE_Contact(in1 := "Input_Data".Load_ScaleA, in2 := "Input_Data".Set_Weight_Gao)
      { S7_Templates := "SrcType := Real" } LT_Contact(in1 := "Input_Data".Load_ScaleA, in2 := #sumGaoSan)
      R_Coil( "DB_TrungGian".Enable_XiloGao )
      R_Coil( "DB_TrungGian".Enable_XiloNgo )
      S_Coil( "DB_TrungGian".Enable_XiloSan )
   END_RUNG
   RUNG wire#w4
      { S7_Templates := "SrcType := Real" } GE_Contact(in1 := "Input_Data".Load_ScaleA, in2 := #sumGaoSan)
      R_Coil( "DB_TrungGian".Enable_XiloGao )
      R_Coil( "DB_TrungGian".Enable_XiloSan )
      S_Coil( "DB_TrungGian".Enable_XiloNgo )
   END_RUNG
   RUNG wire#w1
      { S7_Templates := "SrcType := Real" } LT_Contact(in1 := "Input_Data".Set_Weight_Gao, in2 := "Input_Data".Set_Weight_San)
      wire#w5
      { S7_Templates := "SrcType := Real" } LT_Contact(in1 := "Input_Data".Load_ScaleA, in2 := "Input_Data".Set_Weight_San)
      R_Coil( "DB_TrungGian".Enable_XiloGao )
      R_Coil( "DB_TrungGian".Enable_XiloNgo )
      S_Coil( "DB_TrungGian".Enable_XiloSan )
   END_RUNG
   RUNG wire#w5
      { S7_Templates := "SrcType := Real" } GE_Contact(in1 := "Input_Data".Load_ScaleA, in2 := "Input_Data".Set_Weight_San)
      { S7_Templates := "SrcType := Real" } LT_Contact(in1 := "Input_Data".Load_ScaleA, in2 := #sumGaoSan)
      R_Coil( "DB_TrungGian".Enable_XiloNgo )
      R_Coil( "DB_TrungGian".Enable_XiloSan )
      S_Coil( "DB_TrungGian".Enable_XiloGao )
   END_RUNG
   RUNG wire#w5
      { S7_Templates := "SrcType := Real" } GE_Contact(in1 := "Input_Data".Load_ScaleA, in2 := #sumGaoSan)
      R_Coil( "DB_TrungGian".Enable_XiloGao )
      R_Coil( "DB_TrungGian".Enable_XiloSan )
      S_Coil( "DB_TrungGian".Enable_XiloNgo )
   END_RUNG
   // the same network as SCL:
   #_w1 := "M_Auto_Motor_Tai" AND NOT "Input".Ss_ScalesA AND ("Input_Data".Set_Weight_Gao >= "Input_Data".Set_Weight_Ngo);
   #_w2 := #_w1 AND ("Input_Data".Set_Weight_Gao >= "Input_Data".Set_Weight_San);
   #_w3 := #_w2 AND ("Input_Data".Set_Weight_Ngo >= "Input_Data".Set_Weight_San);
   IF #_w3 AND ("Input_Data".Load_ScaleA < "Input_Data".Set_Weight_Gao) THEN
       "DB_TrungGian".Enable_XiloNgo := FALSE;
       "DB_TrungGian".Enable_XiloSan := FALSE;
       "DB_TrungGian".Enable_XiloGao := TRUE;
   END_IF;
   IF #_w3 AND ("Input_Data".Load_ScaleA >= "Input_Data".Set_Weight_Gao) AND ("Input_Data".Load_ScaleA < #sumGaoNgo) THEN
       "DB_TrungGian".Enable_XiloGao := FALSE;
       "DB_TrungGian".Enable_XiloSan := FALSE;
       "DB_TrungGian".Enable_XiloNgo := TRUE;
   END_IF;
   IF #_w3 AND ("Input_Data".Load_ScaleA >= #sumGaoNgo) THEN
       "DB_TrungGian".Enable_XiloNgo := FALSE;
       "DB_TrungGian".Enable_XiloGao := FALSE;
       "DB_TrungGian".Enable_XiloSan := TRUE;
   END_IF;
   #_w4 := #_w2 AND ("Input_Data".Set_Weight_Ngo < "Input_Data".Set_Weight_San);
   IF #_w4 AND ("Input_Data".Load_ScaleA < "Input_Data".Set_Weight_Gao) THEN
       "DB_TrungGian".Enable_XiloNgo := FALSE;
       "DB_TrungGian".Enable_XiloSan := FALSE;
       "DB_TrungGian".Enable_XiloGao := TRUE;
   END_IF;
   IF #_w4 AND ("Input_Data".Load_ScaleA >= "Input_Data".Set_Weight_Gao) AND ("Input_Data".Load_ScaleA < #sumGaoSan) THEN
       "DB_TrungGian".Enable_XiloGao := FALSE;
       "DB_TrungGian".Enable_XiloNgo := FALSE;
       "DB_TrungGian".Enable_XiloSan := TRUE;
   END_IF;
   IF #_w4 AND ("Input_Data".Load_ScaleA >= #sumGaoSan) THEN
       "DB_TrungGian".Enable_XiloGao := FALSE;
       "DB_TrungGian".Enable_XiloSan := FALSE;
       "DB_TrungGian".Enable_XiloNgo := TRUE;
   END_IF;
   #_w5 := #_w1 AND ("Input_Data".Set_Weight_Gao < "Input_Data".Set_Weight_San);
   IF #_w5 AND ("Input_Data".Load_ScaleA < "Input_Data".Set_Weight_San) THEN
       "DB_TrungGian".Enable_XiloGao := FALSE;
       "DB_TrungGian".Enable_XiloNgo := FALSE;
       "DB_TrungGian".Enable_XiloSan := TRUE;
   END_IF;
   IF #_w5 AND ("Input_Data".Load_ScaleA >= "Input_Data".Set_Weight_San) AND ("Input_Data".Load_ScaleA < #sumGaoSan) THEN
       "DB_TrungGian".Enable_XiloNgo := FALSE;
       "DB_TrungGian".Enable_XiloSan := FALSE;
       "DB_TrungGian".Enable_XiloGao := TRUE;
   END_IF;
   IF #_w5 AND ("Input_Data".Load_ScaleA >= #sumGaoSan) THEN
       "DB_TrungGian".Enable_XiloGao := FALSE;
       "DB_TrungGian".Enable_XiloSan := FALSE;
       "DB_TrungGian".Enable_XiloNgo := TRUE;
   END_IF;
END_REGION

REGION Network 5
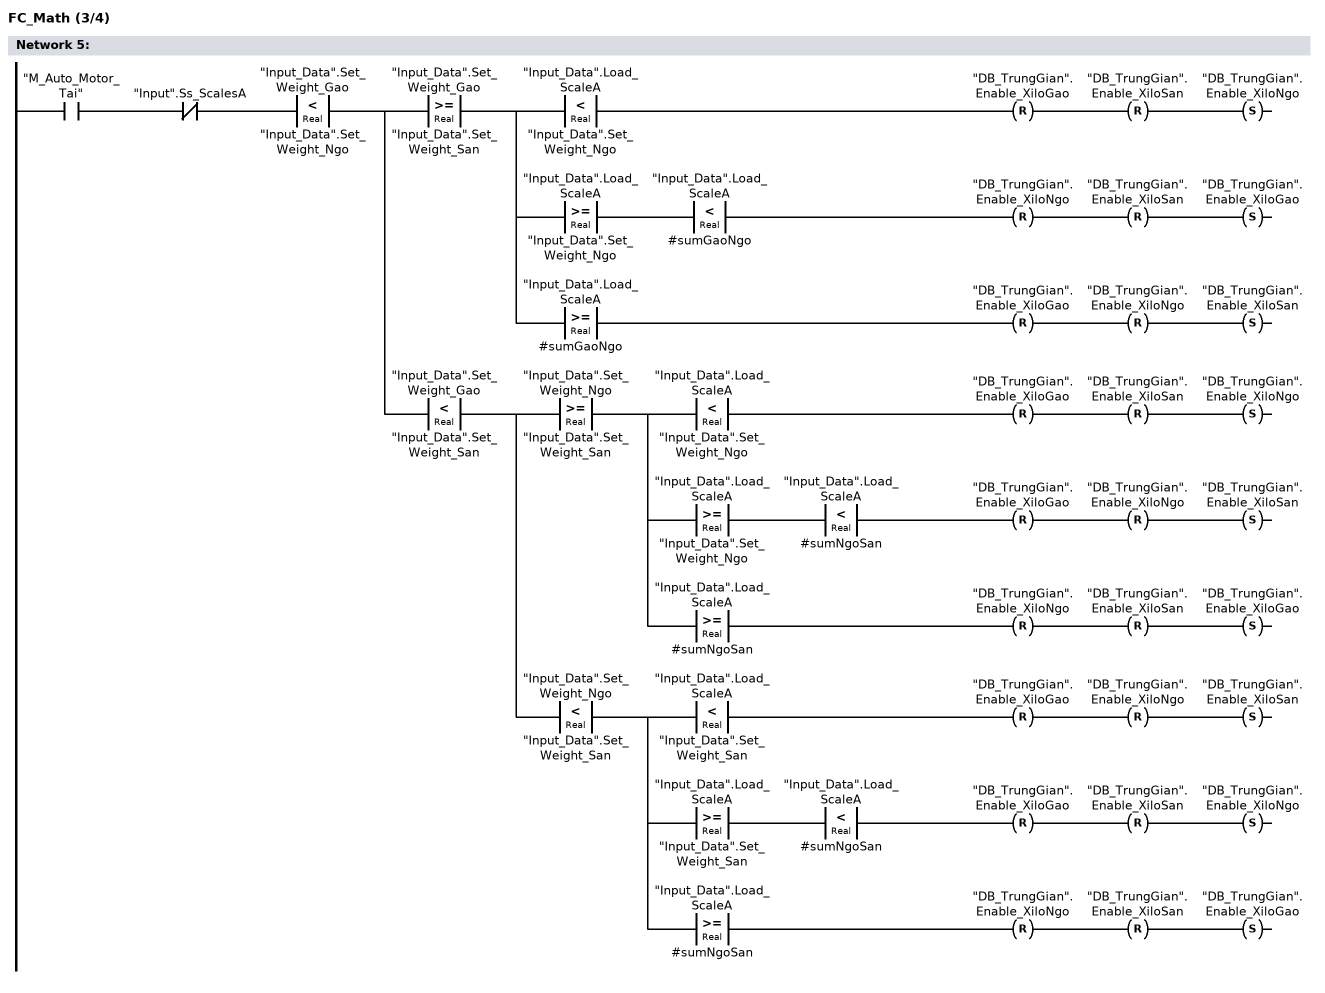
   RUNG wire#powerrail
      Contact( "M_Auto_Motor_Tai" )
      I_Contact( "Input".Ss_ScalesA )
      { S7_Templates := "SrcType := Real" } LT_Contact(in1 := "Input_Data".Set_Weight_Gao, in2 := "Input_Data".Set_Weight_Ngo)
      wire#w1
      { S7_Templates := "SrcType := Real" } GE_Contact(in1 := "Input_Data".Set_Weight_Gao, in2 := "Input_Data".Set_Weight_San)
      wire#w2
      { S7_Templates := "SrcType := Real" } LT_Contact(in1 := "Input_Data".Load_ScaleA, in2 := "Input_Data".Set_Weight_Ngo)
      R_Coil( "DB_TrungGian".Enable_XiloGao )
      R_Coil( "DB_TrungGian".Enable_XiloSan )
      S_Coil( "DB_TrungGian".Enable_XiloNgo )
   END_RUNG
   RUNG wire#w2
      { S7_Templates := "SrcType := Real" } GE_Contact(in1 := "Input_Data".Load_ScaleA, in2 := "Input_Data".Set_Weight_Ngo)
      { S7_Templates := "SrcType := Real" } LT_Contact(in1 := "Input_Data".Load_ScaleA, in2 := #sumGaoNgo)
      R_Coil( "DB_TrungGian".Enable_XiloNgo )
      R_Coil( "DB_TrungGian".Enable_XiloSan )
      S_Coil( "DB_TrungGian".Enable_XiloGao )
   END_RUNG
   RUNG wire#w2
      { S7_Templates := "SrcType := Real" } GE_Contact(in1 := "Input_Data".Load_ScaleA, in2 := #sumGaoNgo)
      R_Coil( "DB_TrungGian".Enable_XiloGao )
      R_Coil( "DB_TrungGian".Enable_XiloNgo )
      S_Coil( "DB_TrungGian".Enable_XiloSan )
   END_RUNG
   RUNG wire#w1
      { S7_Templates := "SrcType := Real" } LT_Contact(in1 := "Input_Data".Set_Weight_Gao, in2 := "Input_Data".Set_Weight_San)
      wire#w3
      { S7_Templates := "SrcType := Real" } GE_Contact(in1 := "Input_Data".Set_Weight_Ngo, in2 := "Input_Data".Set_Weight_San)
      wire#w4
      { S7_Templates := "SrcType := Real" } LT_Contact(in1 := "Input_Data".Load_ScaleA, in2 := "Input_Data".Set_Weight_Ngo)
      R_Coil( "DB_TrungGian".Enable_XiloGao )
      R_Coil( "DB_TrungGian".Enable_XiloSan )
      S_Coil( "DB_TrungGian".Enable_XiloNgo )
   END_RUNG
   RUNG wire#w4
      { S7_Templates := "SrcType := Real" } GE_Contact(in1 := "Input_Data".Load_ScaleA, in2 := "Input_Data".Set_Weight_Ngo)
      { S7_Templates := "SrcType := Real" } LT_Contact(in1 := "Input_Data".Load_ScaleA, in2 := #sumNgoSan)
      R_Coil( "DB_TrungGian".Enable_XiloGao )
      R_Coil( "DB_TrungGian".Enable_XiloNgo )
      S_Coil( "DB_TrungGian".Enable_XiloSan )
   END_RUNG
   RUNG wire#w4
      { S7_Templates := "SrcType := Real" } GE_Contact(in1 := "Input_Data".Load_ScaleA, in2 := #sumNgoSan)
      R_Coil( "DB_TrungGian".Enable_XiloNgo )
      R_Coil( "DB_TrungGian".Enable_XiloSan )
      S_Coil( "DB_TrungGian".Enable_XiloGao )
   END_RUNG
   RUNG wire#w3
      { S7_Templates := "SrcType := Real" } LT_Contact(in1 := "Input_Data".Set_Weight_Ngo, in2 := "Input_Data".Set_Weight_San)
      wire#w5
      { S7_Templates := "SrcType := Real" } LT_Contact(in1 := "Input_Data".Load_ScaleA, in2 := "Input_Data".Set_Weight_San)
      R_Coil( "DB_TrungGian".Enable_XiloGao )
      R_Coil( "DB_TrungGian".Enable_XiloNgo )
      S_Coil( "DB_TrungGian".Enable_XiloSan )
   END_RUNG
   RUNG wire#w5
      { S7_Templates := "SrcType := Real" } GE_Contact(in1 := "Input_Data".Load_ScaleA, in2 := "Input_Data".Set_Weight_San)
      { S7_Templates := "SrcType := Real" } LT_Contact(in1 := "Input_Data".Load_ScaleA, in2 := #sumNgoSan)
      R_Coil( "DB_TrungGian".Enable_XiloGao )
      R_Coil( "DB_TrungGian".Enable_XiloSan )
      S_Coil( "DB_TrungGian".Enable_XiloNgo )
   END_RUNG
   RUNG wire#w5
      { S7_Templates := "SrcType := Real" } GE_Contact(in1 := "Input_Data".Load_ScaleA, in2 := #sumNgoSan)
      R_Coil( "DB_TrungGian".Enable_XiloNgo )
      R_Coil( "DB_TrungGian".Enable_XiloSan )
      S_Coil( "DB_TrungGian".Enable_XiloGao )
   END_RUNG
   // the same network as SCL:
   #_w1 := "M_Auto_Motor_Tai" AND NOT "Input".Ss_ScalesA AND ("Input_Data".Set_Weight_Gao < "Input_Data".Set_Weight_Ngo);
   #_w2 := #_w1 AND ("Input_Data".Set_Weight_Gao >= "Input_Data".Set_Weight_San);
   IF #_w2 AND ("Input_Data".Load_ScaleA < "Input_Data".Set_Weight_Ngo) THEN
       "DB_TrungGian".Enable_XiloGao := FALSE;
       "DB_TrungGian".Enable_XiloSan := FALSE;
       "DB_TrungGian".Enable_XiloNgo := TRUE;
   END_IF;
   IF #_w2 AND ("Input_Data".Load_ScaleA >= "Input_Data".Set_Weight_Ngo) AND ("Input_Data".Load_ScaleA < #sumGaoNgo) THEN
       "DB_TrungGian".Enable_XiloNgo := FALSE;
       "DB_TrungGian".Enable_XiloSan := FALSE;
       "DB_TrungGian".Enable_XiloGao := TRUE;
   END_IF;
   IF #_w2 AND ("Input_Data".Load_ScaleA >= #sumGaoNgo) THEN
       "DB_TrungGian".Enable_XiloGao := FALSE;
       "DB_TrungGian".Enable_XiloNgo := FALSE;
       "DB_TrungGian".Enable_XiloSan := TRUE;
   END_IF;
   #_w3 := #_w1 AND ("Input_Data".Set_Weight_Gao < "Input_Data".Set_Weight_San);
   #_w4 := #_w3 AND ("Input_Data".Set_Weight_Ngo >= "Input_Data".Set_Weight_San);
   IF #_w4 AND ("Input_Data".Load_ScaleA < "Input_Data".Set_Weight_Ngo) THEN
       "DB_TrungGian".Enable_XiloGao := FALSE;
       "DB_TrungGian".Enable_XiloSan := FALSE;
       "DB_TrungGian".Enable_XiloNgo := TRUE;
   END_IF;
   IF #_w4 AND ("Input_Data".Load_ScaleA >= "Input_Data".Set_Weight_Ngo) AND ("Input_Data".Load_ScaleA < #sumNgoSan) THEN
       "DB_TrungGian".Enable_XiloGao := FALSE;
       "DB_TrungGian".Enable_XiloNgo := FALSE;
       "DB_TrungGian".Enable_XiloSan := TRUE;
   END_IF;
   IF #_w4 AND ("Input_Data".Load_ScaleA >= #sumNgoSan) THEN
       "DB_TrungGian".Enable_XiloNgo := FALSE;
       "DB_TrungGian".Enable_XiloSan := FALSE;
       "DB_TrungGian".Enable_XiloGao := TRUE;
   END_IF;
   #_w5 := #_w3 AND ("Input_Data".Set_Weight_Ngo < "Input_Data".Set_Weight_San);
   IF #_w5 AND ("Input_Data".Load_ScaleA < "Input_Data".Set_Weight_San) THEN
       "DB_TrungGian".Enable_XiloGao := FALSE;
       "DB_TrungGian".Enable_XiloNgo := FALSE;
       "DB_TrungGian".Enable_XiloSan := TRUE;
   END_IF;
   IF #_w5 AND ("Input_Data".Load_ScaleA >= "Input_Data".Set_Weight_San) AND ("Input_Data".Load_ScaleA < #sumNgoSan) THEN
       "DB_TrungGian".Enable_XiloGao := FALSE;
       "DB_TrungGian".Enable_XiloSan := FALSE;
       "DB_TrungGian".Enable_XiloNgo := TRUE;
   END_IF;
   IF #_w5 AND ("Input_Data".Load_ScaleA >= #sumNgoSan) THEN
       "DB_TrungGian".Enable_XiloNgo := FALSE;
       "DB_TrungGian".Enable_XiloSan := FALSE;
       "DB_TrungGian".Enable_XiloGao := TRUE;
   END_IF;
END_REGION

REGION Network 6: cân A cân xong, tiếp tục so sánh giá trị cân n.liệu đầu vào cân B
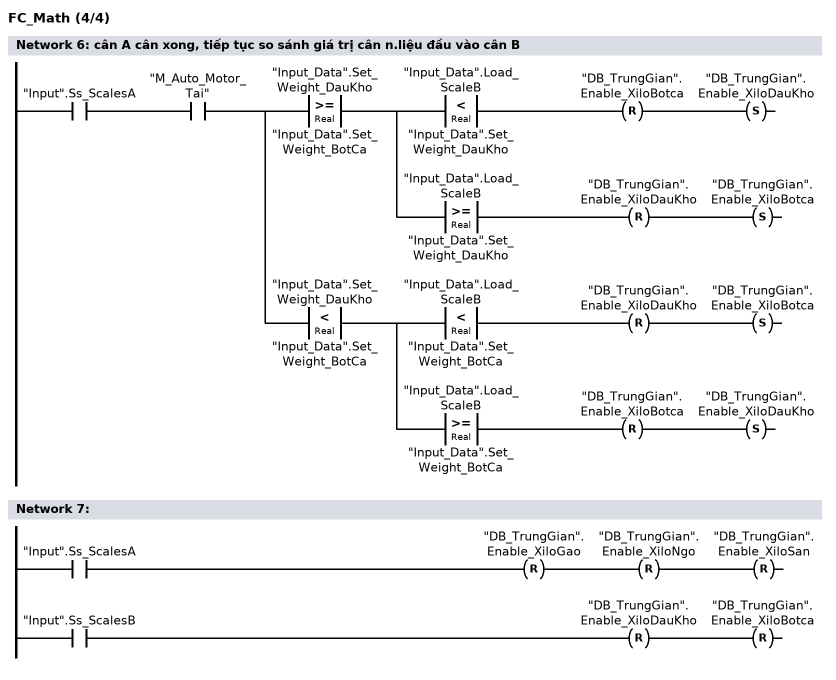
   RUNG wire#powerrail
      Contact( "Input".Ss_ScalesA )
      Contact( "M_Auto_Motor_Tai" )
      wire#w1
      { S7_Templates := "SrcType := Real" } GE_Contact(in1 := "Input_Data".Set_Weight_DauKho, in2 := "Input_Data".Set_Weight_BotCa)
      wire#w2
      { S7_Templates := "SrcType := Real" } LT_Contact(in1 := "Input_Data".Load_ScaleB, in2 := "Input_Data".Set_Weight_DauKho)
      R_Coil( "DB_TrungGian".Enable_XiloBotca )
      S_Coil( "DB_TrungGian".Enable_XiloDauKho )
   END_RUNG
   RUNG wire#w2
      { S7_Templates := "SrcType := Real" } GE_Contact(in1 := "Input_Data".Load_ScaleB, in2 := "Input_Data".Set_Weight_DauKho)
      R_Coil( "DB_TrungGian".Enable_XiloDauKho )
      S_Coil( "DB_TrungGian".Enable_XiloBotca )
   END_RUNG
   RUNG wire#w1
      { S7_Templates := "SrcType := Real" } LT_Contact(in1 := "Input_Data".Set_Weight_DauKho, in2 := "Input_Data".Set_Weight_BotCa)
      wire#w3
      { S7_Templates := "SrcType := Real" } LT_Contact(in1 := "Input_Data".Load_ScaleB, in2 := "Input_Data".Set_Weight_BotCa)
      R_Coil( "DB_TrungGian".Enable_XiloDauKho )
      S_Coil( "DB_TrungGian".Enable_XiloBotca )
   END_RUNG
   RUNG wire#w3
      { S7_Templates := "SrcType := Real" } GE_Contact(in1 := "Input_Data".Load_ScaleB, in2 := "Input_Data".Set_Weight_BotCa)
      R_Coil( "DB_TrungGian".Enable_XiloBotca )
      S_Coil( "DB_TrungGian".Enable_XiloDauKho )
   END_RUNG
   // the same network as SCL:
   #_w1 := "Input".Ss_ScalesA AND "M_Auto_Motor_Tai";
   #_w2 := #_w1 AND ("Input_Data".Set_Weight_DauKho >= "Input_Data".Set_Weight_BotCa);
   IF #_w2 AND ("Input_Data".Load_ScaleB < "Input_Data".Set_Weight_DauKho) THEN
       "DB_TrungGian".Enable_XiloBotca := FALSE;
       "DB_TrungGian".Enable_XiloDauKho := TRUE;
   END_IF;
   IF #_w2 AND ("Input_Data".Load_ScaleB >= "Input_Data".Set_Weight_DauKho) THEN
       "DB_TrungGian".Enable_XiloDauKho := FALSE;
       "DB_TrungGian".Enable_XiloBotca := TRUE;
   END_IF;
   #_w3 := #_w1 AND ("Input_Data".Set_Weight_DauKho < "Input_Data".Set_Weight_BotCa);
   IF #_w3 AND ("Input_Data".Load_ScaleB < "Input_Data".Set_Weight_BotCa) THEN
       "DB_TrungGian".Enable_XiloDauKho := FALSE;
       "DB_TrungGian".Enable_XiloBotca := TRUE;
   END_IF;
   IF #_w3 AND ("Input_Data".Load_ScaleB >= "Input_Data".Set_Weight_BotCa) THEN
       "DB_TrungGian".Enable_XiloBotca := FALSE;
       "DB_TrungGian".Enable_XiloDauKho := TRUE;
   END_IF;
END_REGION

REGION Network 7
   RUNG wire#powerrail
      Contact( "Input".Ss_ScalesA )
      R_Coil( "DB_TrungGian".Enable_XiloGao )
      R_Coil( "DB_TrungGian".Enable_XiloNgo )
      R_Coil( "DB_TrungGian".Enable_XiloSan )
   END_RUNG
   RUNG wire#powerrail
      Contact( "Input".Ss_ScalesB )
      R_Coil( "DB_TrungGian".Enable_XiloDauKho )
      R_Coil( "DB_TrungGian".Enable_XiloBotca )
   END_RUNG
   // the same network as SCL:
   IF "Input".Ss_ScalesA THEN
       "DB_TrungGian".Enable_XiloGao := FALSE;
       "DB_TrungGian".Enable_XiloNgo := FALSE;
       "DB_TrungGian".Enable_XiloSan := FALSE;
   END_IF;
   IF "Input".Ss_ScalesB THEN
       "DB_TrungGian".Enable_XiloDauKho := FALSE;
       "DB_TrungGian".Enable_XiloBotca := FALSE;
   END_IF;
END_REGION
END_FUNCTION

FUNCTION "FC_XiloGao" : Void   // FC6, LAD
{ S7_Optimized_Access := 'TRUE' }
VERSION : 0.1
   VAR_TEMP
      sum1_Xilo : Real;
      sum2_Xilo : Real;
   END_VAR
   VAR_TEMP   // added for the SCL form of the ladder/FBD networks
      _w1 : Bool;
      _w2 : Bool;
   END_VAR
BEGIN

REGION Network 1: K.lượng gạo = a
   // tính 2 giá trị a/3 và 2a/3
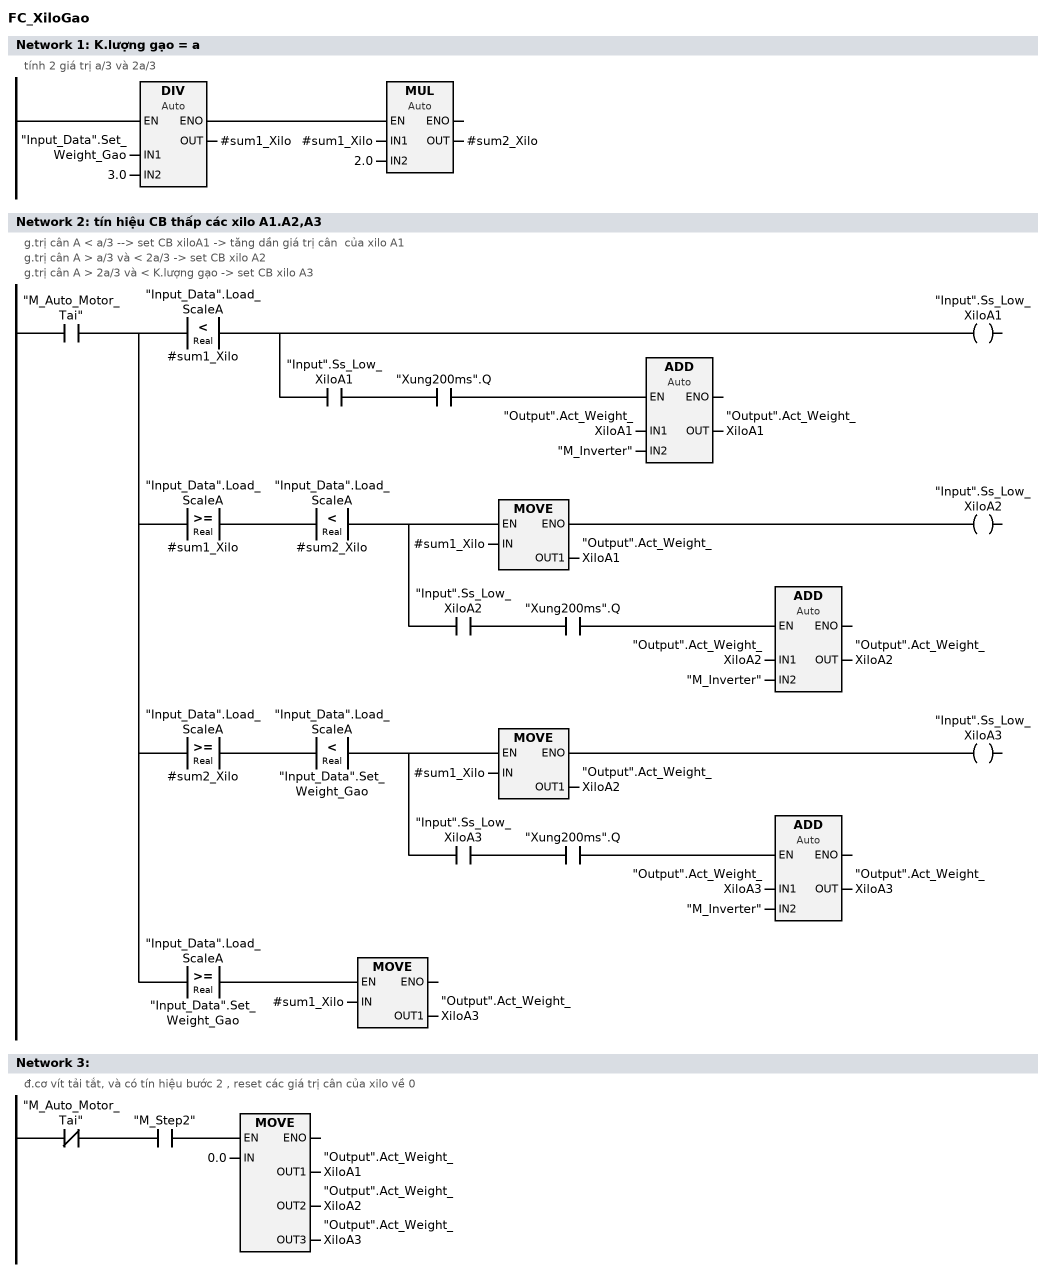
   RUNG wire#powerrail
      Div(in1 := "Input_Data".Set_Weight_Gao, in2 := 3.0, out => #sum1_Xilo)
      Mul(in1 := #sum1_Xilo, in2 := 2.0, out => #sum2_Xilo)
   END_RUNG
   // the same network as SCL:
   #sum1_Xilo := "Input_Data".Set_Weight_Gao / 3.0;
   #sum2_Xilo := #sum1_Xilo * 2.0;
END_REGION

REGION Network 2: tín hiệu CB thấp các xilo A1.A2,A3
   // g.trị cân A < a/3 --> set CB xiloA1 -> tăng dần giá trị cân  của xilo A1
   // g.trị cân A > a/3 và < 2a/3 -> set CB xilo A2
   // g.trị cân A > 2a/3 và < K.lượng gạo -> set CB xilo A3
   RUNG wire#powerrail
      Contact( "M_Auto_Motor_Tai" )
      wire#w1
      { S7_Templates := "SrcType := Real" } LT_Contact(in1 := "Input_Data".Load_ScaleA, in2 := #sum1_Xilo)
      wire#w2
      Coil( "Input".Ss_Low_XiloA1 )
   END_RUNG
   RUNG wire#w2
      Contact( "Input".Ss_Low_XiloA1 )
      Contact( "Xung200ms".Q )
      Add(in1 := "Output".Act_Weight_XiloA1, in2 := "M_Inverter", out => "Output".Act_Weight_XiloA1)
   END_RUNG
   RUNG wire#w1
      { S7_Templates := "SrcType := Real" } GE_Contact(in1 := "Input_Data".Load_ScaleA, in2 := #sum1_Xilo)
      { S7_Templates := "SrcType := Real" } LT_Contact(in1 := "Input_Data".Load_ScaleA, in2 := #sum2_Xilo)
      wire#w3
      Move(in := #sum1_Xilo, out1 => "Output".Act_Weight_XiloA1)
      Coil( "Input".Ss_Low_XiloA2 )
   END_RUNG
   RUNG wire#w3
      Contact( "Input".Ss_Low_XiloA2 )
      Contact( "Xung200ms".Q )
      Add(in1 := "Output".Act_Weight_XiloA2, in2 := "M_Inverter", out => "Output".Act_Weight_XiloA2)
   END_RUNG
   RUNG wire#w1
      { S7_Templates := "SrcType := Real" } GE_Contact(in1 := "Input_Data".Load_ScaleA, in2 := #sum2_Xilo)
      { S7_Templates := "SrcType := Real" } LT_Contact(in1 := "Input_Data".Load_ScaleA, in2 := "Input_Data".Set_Weight_Gao)
      wire#w4
      Move(in := #sum1_Xilo, out1 => "Output".Act_Weight_XiloA2)
      Coil( "Input".Ss_Low_XiloA3 )
   END_RUNG
   RUNG wire#w4
      Contact( "Input".Ss_Low_XiloA3 )
      Contact( "Xung200ms".Q )
      Add(in1 := "Output".Act_Weight_XiloA3, in2 := "M_Inverter", out => "Output".Act_Weight_XiloA3)
   END_RUNG
   RUNG wire#w1
      { S7_Templates := "SrcType := Real" } GE_Contact(in1 := "Input_Data".Load_ScaleA, in2 := "Input_Data".Set_Weight_Gao)
      Move(in := #sum1_Xilo, out1 => "Output".Act_Weight_XiloA3)
   END_RUNG
   // the same network as SCL:
   "Input".Ss_Low_XiloA1 := "M_Auto_Motor_Tai" AND ("Input_Data".Load_ScaleA < #sum1_Xilo);
   IF "Input".Ss_Low_XiloA1 AND "Input".Ss_Low_XiloA1 AND "Xung200ms".Q THEN
       "Output".Act_Weight_XiloA1 := "Output".Act_Weight_XiloA1 + "M_Inverter";
   END_IF;
   #_w1 := "M_Auto_Motor_Tai" AND ("Input_Data".Load_ScaleA >= #sum1_Xilo) AND ("Input_Data".Load_ScaleA < #sum2_Xilo);
   IF #_w1 THEN "Output".Act_Weight_XiloA1 := #sum1_Xilo; END_IF;
   "Input".Ss_Low_XiloA2 := #_w1;
   IF #_w1 AND "Input".Ss_Low_XiloA2 AND "Xung200ms".Q THEN
       "Output".Act_Weight_XiloA2 := "Output".Act_Weight_XiloA2 + "M_Inverter";
   END_IF;
   #_w2 := "M_Auto_Motor_Tai" AND ("Input_Data".Load_ScaleA >= #sum2_Xilo) AND ("Input_Data".Load_ScaleA < "Input_Data".Set_Weight_Gao);
   IF #_w2 THEN "Output".Act_Weight_XiloA2 := #sum1_Xilo; END_IF;
   "Input".Ss_Low_XiloA3 := #_w2;
   IF #_w2 AND "Input".Ss_Low_XiloA3 AND "Xung200ms".Q THEN
       "Output".Act_Weight_XiloA3 := "Output".Act_Weight_XiloA3 + "M_Inverter";
   END_IF;
   IF "M_Auto_Motor_Tai" AND ("Input_Data".Load_ScaleA >= "Input_Data".Set_Weight_Gao) THEN
       "Output".Act_Weight_XiloA3 := #sum1_Xilo;
   END_IF;
END_REGION

REGION Network 3
   // đ.cơ vít tải tắt, và có tín hiệu bước 2 , reset các giá trị cân của xilo về 0
   RUNG wire#powerrail
      I_Contact( "M_Auto_Motor_Tai" )
      Contact( "M_Step2" )
      Move(in := 0.0, out1 => "Output".Act_Weight_XiloA1, out2 => "Output".Act_Weight_XiloA2, out3 => "Output".Act_Weight_XiloA3)
   END_RUNG
   // the same network as SCL:
   IF NOT "M_Auto_Motor_Tai" AND "M_Step2" THEN
       "Output".Act_Weight_XiloA1 := 0.0;
       "Output".Act_Weight_XiloA2 := 0.0;
       "Output".Act_Weight_XiloA3 := 0.0;
   END_IF;
END_REGION
END_FUNCTION

FUNCTION "FC_XiloNgo" : Void   // FC7, LAD
{ S7_Optimized_Access := 'TRUE' }
VERSION : 0.1
   VAR_TEMP
      sum1_Xilo : Real;
      sum2_Xilo : Real;
      sum3_Xilo : Real;
      "1" : Real;
      "2" : Real;
      "3" : Real;
      "4" : Real;
   END_VAR
   VAR_TEMP   // added for the SCL form of the ladder/FBD networks
      _w1 : Bool;
      _w2 : Bool;
      _w3 : Bool;
   END_VAR
BEGIN

REGION Network 1: K.lượng Ngô = b
   // Tính các giá trị b/4 , 2b/4, 3b/4
   // Tính các giá trị a+b/4 , a+2b/4 , a+3b/4 , a+b
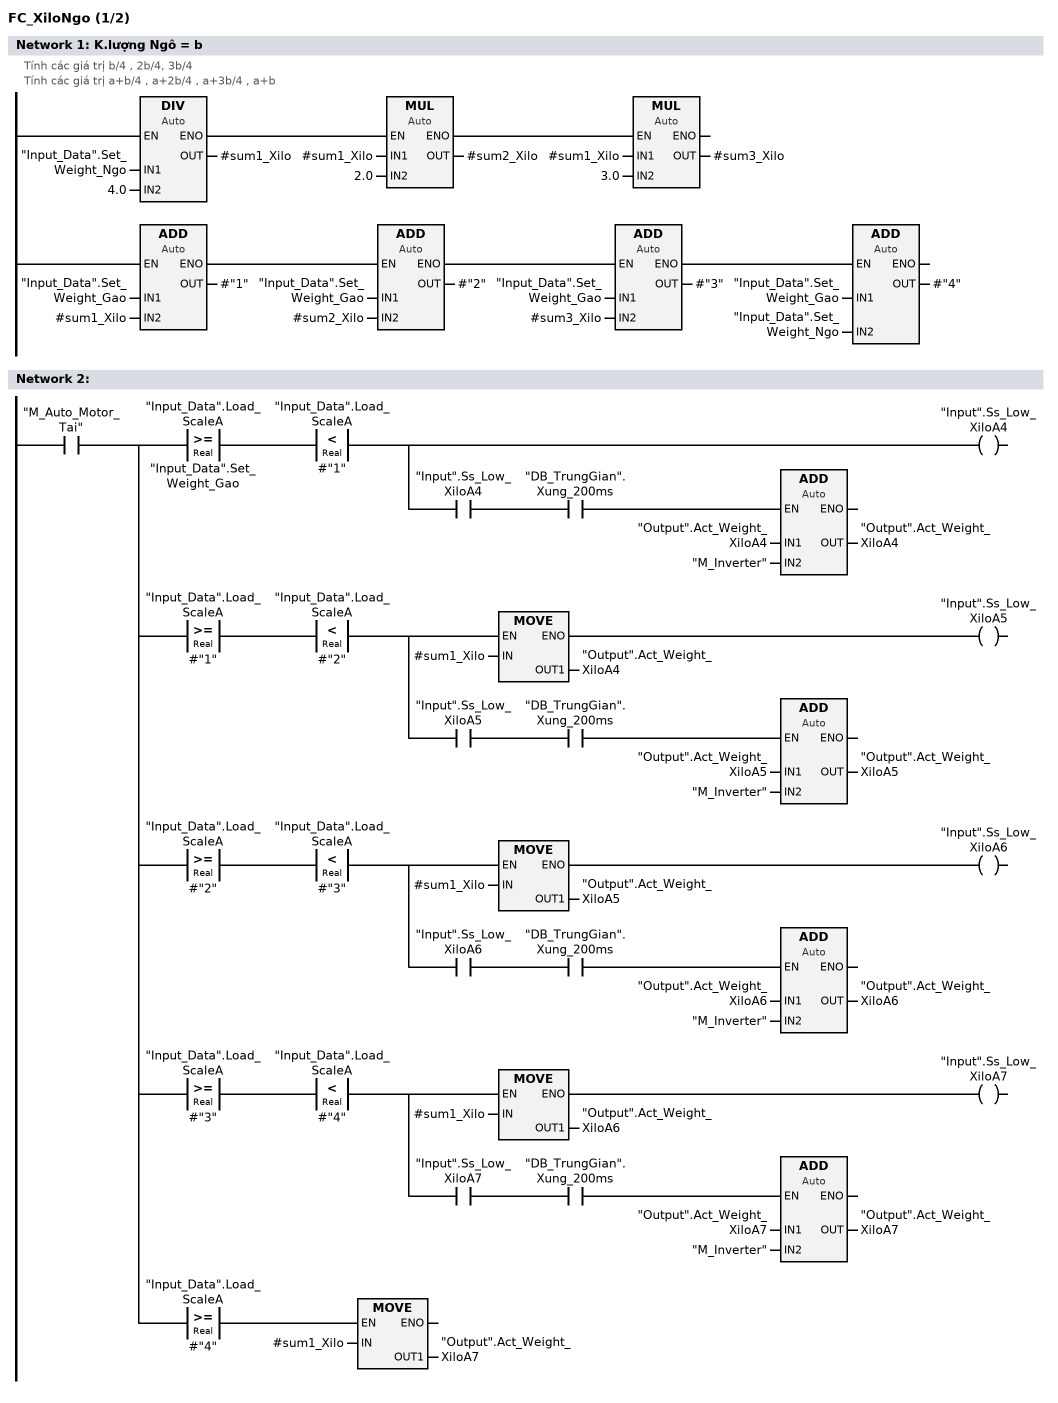
   RUNG wire#powerrail
      Div(in1 := "Input_Data".Set_Weight_Ngo, in2 := 4.0, out => #sum1_Xilo)
      Mul(in1 := #sum1_Xilo, in2 := 2.0, out => #sum2_Xilo)
      Mul(in1 := #sum1_Xilo, in2 := 3.0, out => #sum3_Xilo)
   END_RUNG
   RUNG wire#powerrail
      Add(in1 := "Input_Data".Set_Weight_Gao, in2 := #sum1_Xilo, out => #"1")
      Add(in1 := "Input_Data".Set_Weight_Gao, in2 := #sum2_Xilo, out => #"2")
      Add(in1 := "Input_Data".Set_Weight_Gao, in2 := #sum3_Xilo, out => #"3")
      Add(in1 := "Input_Data".Set_Weight_Gao, in2 := "Input_Data".Set_Weight_Ngo, out => #"4")
   END_RUNG
   // the same network as SCL:
   #sum1_Xilo := "Input_Data".Set_Weight_Ngo / 4.0;
   #sum2_Xilo := #sum1_Xilo * 2.0;
   #sum3_Xilo := #sum1_Xilo * 3.0;
   #"1" := "Input_Data".Set_Weight_Gao + #sum1_Xilo;
   #"2" := "Input_Data".Set_Weight_Gao + #sum2_Xilo;
   #"3" := "Input_Data".Set_Weight_Gao + #sum3_Xilo;
   #"4" := "Input_Data".Set_Weight_Gao + "Input_Data".Set_Weight_Ngo;
END_REGION

REGION Network 2
   RUNG wire#powerrail
      Contact( "M_Auto_Motor_Tai" )
      wire#w1
      { S7_Templates := "SrcType := Real" } GE_Contact(in1 := "Input_Data".Load_ScaleA, in2 := "Input_Data".Set_Weight_Gao)
      { S7_Templates := "SrcType := Real" } LT_Contact(in1 := "Input_Data".Load_ScaleA, in2 := #"1")
      wire#w2
      Coil( "Input".Ss_Low_XiloA4 )
   END_RUNG
   RUNG wire#w2
      Contact( "Input".Ss_Low_XiloA4 )
      Contact( "DB_TrungGian".Xung_200ms )
      Add(in1 := "Output".Act_Weight_XiloA4, in2 := "M_Inverter", out => "Output".Act_Weight_XiloA4)
   END_RUNG
   RUNG wire#w1
      { S7_Templates := "SrcType := Real" } GE_Contact(in1 := "Input_Data".Load_ScaleA, in2 := #"1")
      { S7_Templates := "SrcType := Real" } LT_Contact(in1 := "Input_Data".Load_ScaleA, in2 := #"2")
      wire#w3
      Move(in := #sum1_Xilo, out1 => "Output".Act_Weight_XiloA4)
      Coil( "Input".Ss_Low_XiloA5 )
   END_RUNG
   RUNG wire#w3
      Contact( "Input".Ss_Low_XiloA5 )
      Contact( "DB_TrungGian".Xung_200ms )
      Add(in1 := "Output".Act_Weight_XiloA5, in2 := "M_Inverter", out => "Output".Act_Weight_XiloA5)
   END_RUNG
   RUNG wire#w1
      { S7_Templates := "SrcType := Real" } GE_Contact(in1 := "Input_Data".Load_ScaleA, in2 := #"2")
      { S7_Templates := "SrcType := Real" } LT_Contact(in1 := "Input_Data".Load_ScaleA, in2 := #"3")
      wire#w4
      Move(in := #sum1_Xilo, out1 => "Output".Act_Weight_XiloA5)
      Coil( "Input".Ss_Low_XiloA6 )
   END_RUNG
   RUNG wire#w4
      Contact( "Input".Ss_Low_XiloA6 )
      Contact( "DB_TrungGian".Xung_200ms )
      Add(in1 := "Output".Act_Weight_XiloA6, in2 := "M_Inverter", out => "Output".Act_Weight_XiloA6)
   END_RUNG
   RUNG wire#w1
      { S7_Templates := "SrcType := Real" } GE_Contact(in1 := "Input_Data".Load_ScaleA, in2 := #"3")
      { S7_Templates := "SrcType := Real" } LT_Contact(in1 := "Input_Data".Load_ScaleA, in2 := #"4")
      wire#w5
      Move(in := #sum1_Xilo, out1 => "Output".Act_Weight_XiloA6)
      Coil( "Input".Ss_Low_XiloA7 )
   END_RUNG
   RUNG wire#w5
      Contact( "Input".Ss_Low_XiloA7 )
      Contact( "DB_TrungGian".Xung_200ms )
      Add(in1 := "Output".Act_Weight_XiloA7, in2 := "M_Inverter", out => "Output".Act_Weight_XiloA7)
   END_RUNG
   RUNG wire#w1
      { S7_Templates := "SrcType := Real" } GE_Contact(in1 := "Input_Data".Load_ScaleA, in2 := #"4")
      Move(in := #sum1_Xilo, out1 => "Output".Act_Weight_XiloA7)
   END_RUNG
   // the same network as SCL:
   "Input".Ss_Low_XiloA4 := "M_Auto_Motor_Tai" AND ("Input_Data".Load_ScaleA >= "Input_Data".Set_Weight_Gao) AND ("Input_Data".Load_ScaleA < #"1");
   IF "Input".Ss_Low_XiloA4 AND "Input".Ss_Low_XiloA4 AND "DB_TrungGian".Xung_200ms THEN
       "Output".Act_Weight_XiloA4 := "Output".Act_Weight_XiloA4 + "M_Inverter";
   END_IF;
   #_w1 := "M_Auto_Motor_Tai" AND ("Input_Data".Load_ScaleA >= #"1") AND ("Input_Data".Load_ScaleA < #"2");
   IF #_w1 THEN "Output".Act_Weight_XiloA4 := #sum1_Xilo; END_IF;
   "Input".Ss_Low_XiloA5 := #_w1;
   IF #_w1 AND "Input".Ss_Low_XiloA5 AND "DB_TrungGian".Xung_200ms THEN
       "Output".Act_Weight_XiloA5 := "Output".Act_Weight_XiloA5 + "M_Inverter";
   END_IF;
   #_w2 := "M_Auto_Motor_Tai" AND ("Input_Data".Load_ScaleA >= #"2") AND ("Input_Data".Load_ScaleA < #"3");
   IF #_w2 THEN "Output".Act_Weight_XiloA5 := #sum1_Xilo; END_IF;
   "Input".Ss_Low_XiloA6 := #_w2;
   IF #_w2 AND "Input".Ss_Low_XiloA6 AND "DB_TrungGian".Xung_200ms THEN
       "Output".Act_Weight_XiloA6 := "Output".Act_Weight_XiloA6 + "M_Inverter";
   END_IF;
   #_w3 := "M_Auto_Motor_Tai" AND ("Input_Data".Load_ScaleA >= #"3") AND ("Input_Data".Load_ScaleA < #"4");
   IF #_w3 THEN "Output".Act_Weight_XiloA6 := #sum1_Xilo; END_IF;
   "Input".Ss_Low_XiloA7 := #_w3;
   IF #_w3 AND "Input".Ss_Low_XiloA7 AND "DB_TrungGian".Xung_200ms THEN
       "Output".Act_Weight_XiloA7 := "Output".Act_Weight_XiloA7 + "M_Inverter";
   END_IF;
   IF "M_Auto_Motor_Tai" AND ("Input_Data".Load_ScaleA >= #"4") THEN
       "Output".Act_Weight_XiloA7 := #sum1_Xilo;
   END_IF;
END_REGION

REGION Network 3
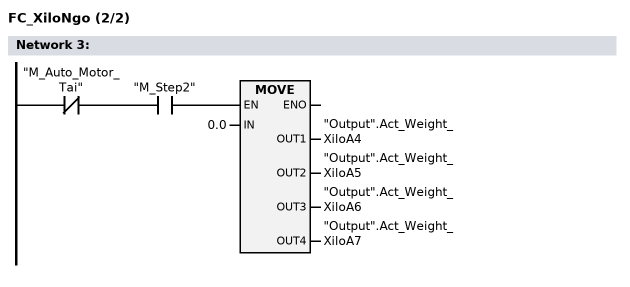
   RUNG wire#powerrail
      I_Contact( "M_Auto_Motor_Tai" )
      Contact( "M_Step2" )
      Move(in := 0.0, out1 => "Output".Act_Weight_XiloA4, out2 => "Output".Act_Weight_XiloA5, out3 => "Output".Act_Weight_XiloA6, out4 => "Output".Act_Weight_XiloA7)
   END_RUNG
   // the same network as SCL:
   IF NOT "M_Auto_Motor_Tai" AND "M_Step2" THEN
       "Output".Act_Weight_XiloA4 := 0.0;
       "Output".Act_Weight_XiloA5 := 0.0;
       "Output".Act_Weight_XiloA6 := 0.0;
       "Output".Act_Weight_XiloA7 := 0.0;
   END_IF;
END_REGION
END_FUNCTION

FUNCTION "FC_XiloSan" : Void   // FC8, LAD
{ S7_Optimized_Access := 'TRUE' }
VERSION : 0.1
   VAR_TEMP
      sum1_Xilo : Real;
      "1" : Real;
      "0" : Real;
   END_VAR
   VAR_TEMP   // added for the SCL form of the ladder/FBD networks
      _w1 : Bool;
   END_VAR
BEGIN

REGION Network 1: k.lượng sắn =c
   // tính các giá trị c/2 , a+b , a+ b + c/2
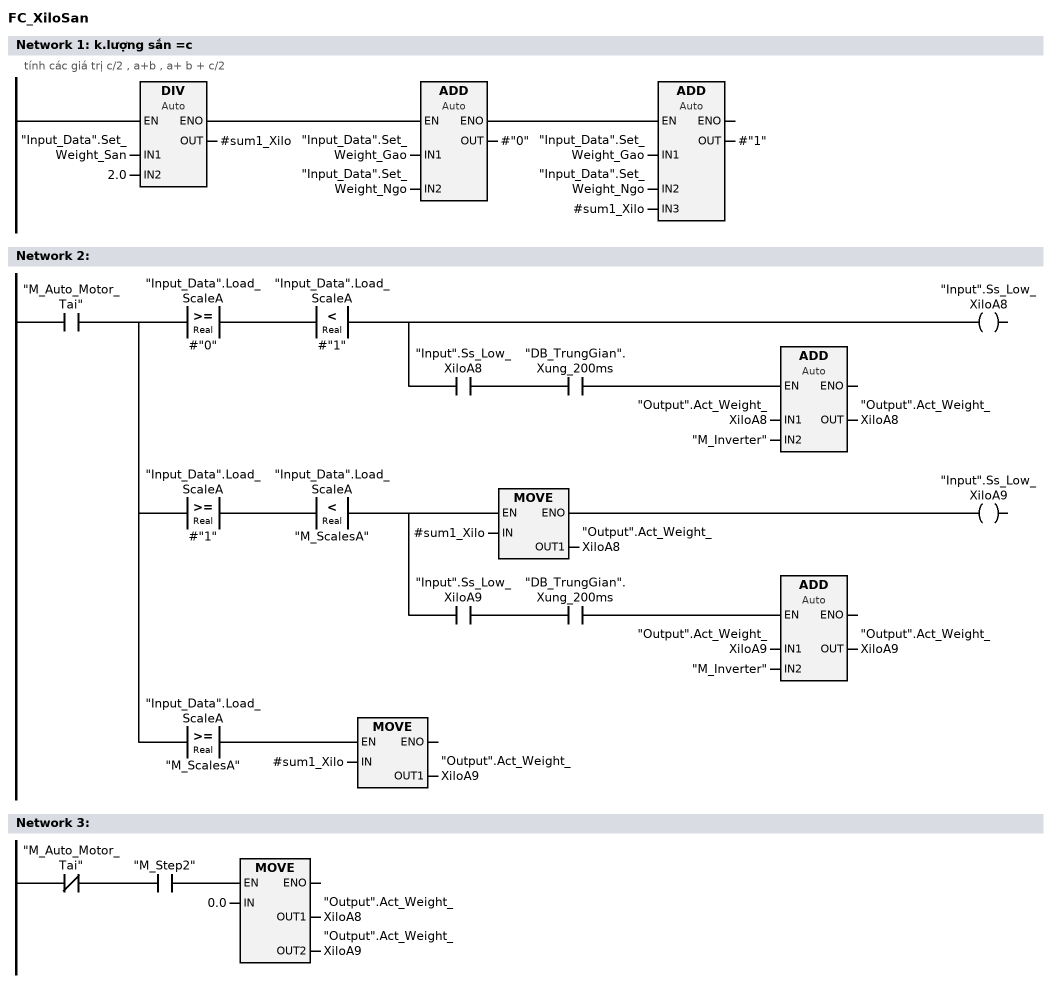
   RUNG wire#powerrail
      Div(in1 := "Input_Data".Set_Weight_San, in2 := 2.0, out => #sum1_Xilo)
      Add(in1 := "Input_Data".Set_Weight_Gao, in2 := "Input_Data".Set_Weight_Ngo, out => #"0")
      Add(in1 := "Input_Data".Set_Weight_Gao, in2 := "Input_Data".Set_Weight_Ngo, in3 := #sum1_Xilo, out => #"1")
   END_RUNG
   // the same network as SCL:
   #sum1_Xilo := "Input_Data".Set_Weight_San / 2.0;
   #"0" := "Input_Data".Set_Weight_Gao + "Input_Data".Set_Weight_Ngo;
   #"1" := "Input_Data".Set_Weight_Gao + "Input_Data".Set_Weight_Ngo + #sum1_Xilo;
END_REGION

REGION Network 2
   RUNG wire#powerrail
      Contact( "M_Auto_Motor_Tai" )
      wire#w1
      { S7_Templates := "SrcType := Real" } GE_Contact(in1 := "Input_Data".Load_ScaleA, in2 := #"0")
      { S7_Templates := "SrcType := Real" } LT_Contact(in1 := "Input_Data".Load_ScaleA, in2 := #"1")
      wire#w2
      Coil( "Input".Ss_Low_XiloA8 )
   END_RUNG
   RUNG wire#w2
      Contact( "Input".Ss_Low_XiloA8 )
      Contact( "DB_TrungGian".Xung_200ms )
      Add(in1 := "Output".Act_Weight_XiloA8, in2 := "M_Inverter", out => "Output".Act_Weight_XiloA8)
   END_RUNG
   RUNG wire#w1
      { S7_Templates := "SrcType := Real" } GE_Contact(in1 := "Input_Data".Load_ScaleA, in2 := #"1")
      { S7_Templates := "SrcType := Real" } LT_Contact(in1 := "Input_Data".Load_ScaleA, in2 := "M_ScalesA")
      wire#w3
      Move(in := #sum1_Xilo, out1 => "Output".Act_Weight_XiloA8)
      Coil( "Input".Ss_Low_XiloA9 )
   END_RUNG
   RUNG wire#w3
      Contact( "Input".Ss_Low_XiloA9 )
      Contact( "DB_TrungGian".Xung_200ms )
      Add(in1 := "Output".Act_Weight_XiloA9, in2 := "M_Inverter", out => "Output".Act_Weight_XiloA9)
   END_RUNG
   RUNG wire#w1
      { S7_Templates := "SrcType := Real" } GE_Contact(in1 := "Input_Data".Load_ScaleA, in2 := "M_ScalesA")
      Move(in := #sum1_Xilo, out1 => "Output".Act_Weight_XiloA9)
   END_RUNG
   // the same network as SCL:
   "Input".Ss_Low_XiloA8 := "M_Auto_Motor_Tai" AND ("Input_Data".Load_ScaleA >= #"0") AND ("Input_Data".Load_ScaleA < #"1");
   IF "Input".Ss_Low_XiloA8 AND "Input".Ss_Low_XiloA8 AND "DB_TrungGian".Xung_200ms THEN
       "Output".Act_Weight_XiloA8 := "Output".Act_Weight_XiloA8 + "M_Inverter";
   END_IF;
   #_w1 := "M_Auto_Motor_Tai" AND ("Input_Data".Load_ScaleA >= #"1") AND ("Input_Data".Load_ScaleA < "M_ScalesA");
   IF #_w1 THEN "Output".Act_Weight_XiloA8 := #sum1_Xilo; END_IF;
   "Input".Ss_Low_XiloA9 := #_w1;
   IF #_w1 AND "Input".Ss_Low_XiloA9 AND "DB_TrungGian".Xung_200ms THEN
       "Output".Act_Weight_XiloA9 := "Output".Act_Weight_XiloA9 + "M_Inverter";
   END_IF;
   IF "M_Auto_Motor_Tai" AND ("Input_Data".Load_ScaleA >= "M_ScalesA") THEN
       "Output".Act_Weight_XiloA9 := #sum1_Xilo;
   END_IF;
END_REGION

REGION Network 3
   RUNG wire#powerrail
      I_Contact( "M_Auto_Motor_Tai" )
      Contact( "M_Step2" )
      Move(in := 0.0, out1 => "Output".Act_Weight_XiloA8, out2 => "Output".Act_Weight_XiloA9)
   END_RUNG
   // the same network as SCL:
   IF NOT "M_Auto_Motor_Tai" AND "M_Step2" THEN
       "Output".Act_Weight_XiloA8 := 0.0;
       "Output".Act_Weight_XiloA9 := 0.0;
   END_IF;
END_REGION
END_FUNCTION

FUNCTION "FC_XiloDauKho" : Void   // FC9, LAD
{ S7_Optimized_Access := 'TRUE' }
VERSION : 0.1
   VAR_TEMP
      sum1_Xilo : Real;
      sum2_Xilo : Real;
   END_VAR
   VAR_TEMP   // added for the SCL form of the ladder/FBD networks
      _w1 : Bool;
      _w2 : Bool;
      _w3 : Bool;
   END_VAR
BEGIN

REGION Network 1: k.lượng đậu khô = d
   // tính các giá trị d/3 , 2d/3
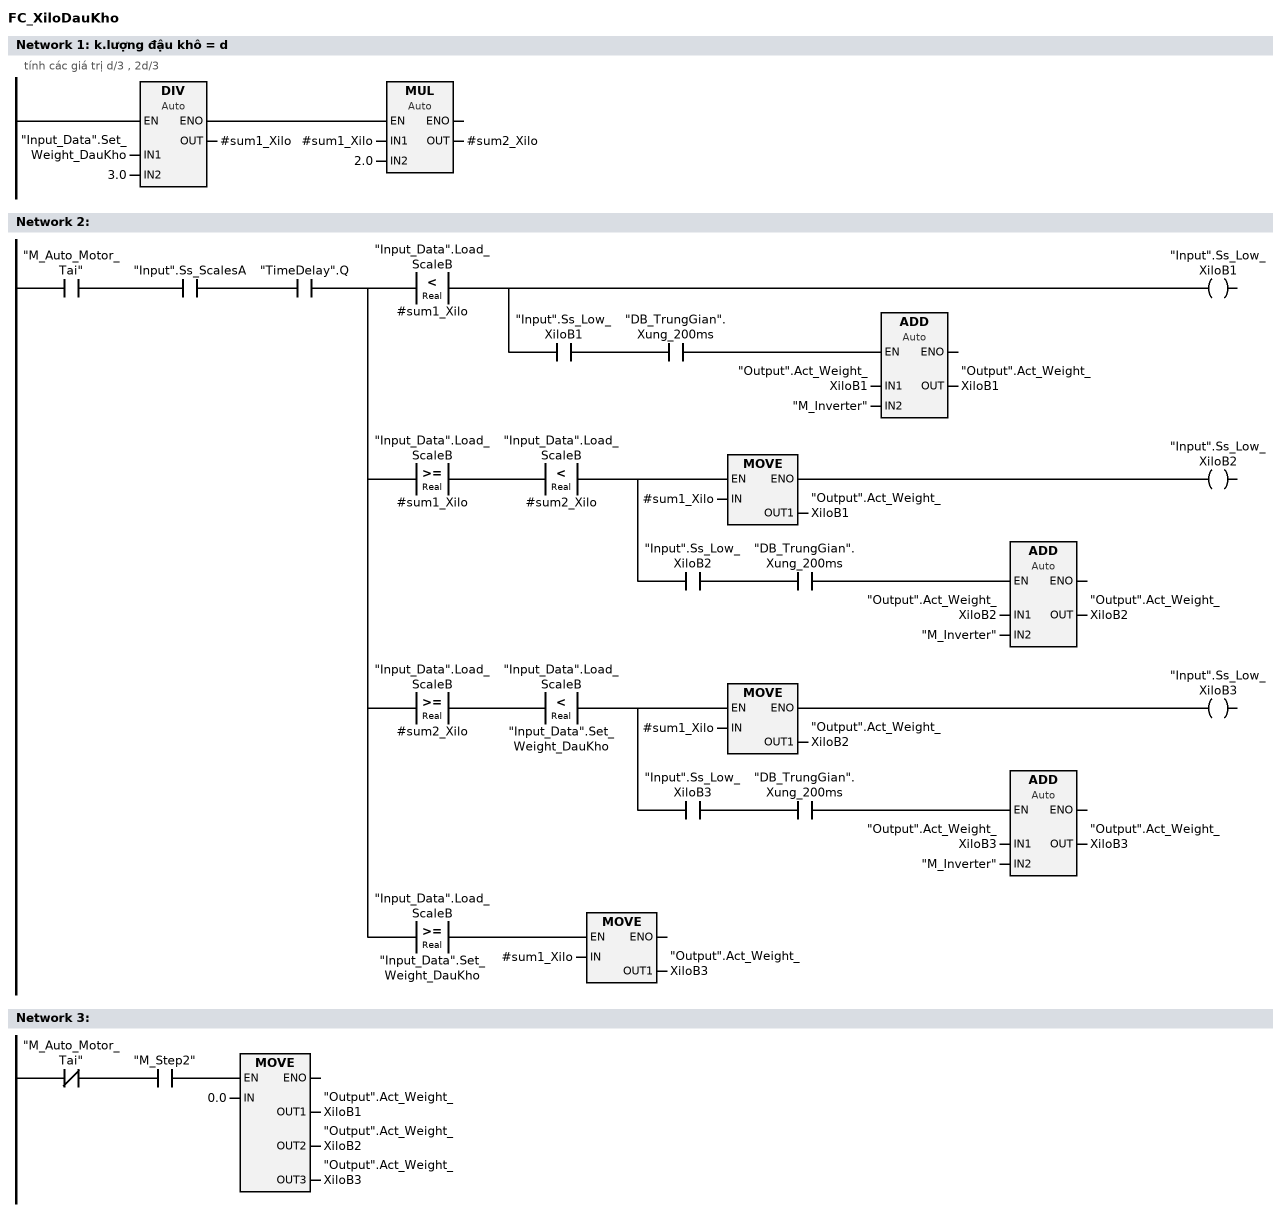
   RUNG wire#powerrail
      Div(in1 := "Input_Data".Set_Weight_DauKho, in2 := 3.0, out => #sum1_Xilo)
      Mul(in1 := #sum1_Xilo, in2 := 2.0, out => #sum2_Xilo)
   END_RUNG
   // the same network as SCL:
   #sum1_Xilo := "Input_Data".Set_Weight_DauKho / 3.0;
   #sum2_Xilo := #sum1_Xilo * 2.0;
END_REGION

REGION Network 2
   RUNG wire#powerrail
      Contact( "M_Auto_Motor_Tai" )
      Contact( "Input".Ss_ScalesA )
      Contact( "TimeDelay".Q )
      wire#w1
      { S7_Templates := "SrcType := Real" } LT_Contact(in1 := "Input_Data".Load_ScaleB, in2 := #sum1_Xilo)
      wire#w2
      Coil( "Input".Ss_Low_XiloB1 )
   END_RUNG
   RUNG wire#w2
      Contact( "Input".Ss_Low_XiloB1 )
      Contact( "DB_TrungGian".Xung_200ms )
      Add(in1 := "Output".Act_Weight_XiloB1, in2 := "M_Inverter", out => "Output".Act_Weight_XiloB1)
   END_RUNG
   RUNG wire#w1
      { S7_Templates := "SrcType := Real" } GE_Contact(in1 := "Input_Data".Load_ScaleB, in2 := #sum1_Xilo)
      { S7_Templates := "SrcType := Real" } LT_Contact(in1 := "Input_Data".Load_ScaleB, in2 := #sum2_Xilo)
      wire#w3
      Move(in := #sum1_Xilo, out1 => "Output".Act_Weight_XiloB1)
      Coil( "Input".Ss_Low_XiloB2 )
   END_RUNG
   RUNG wire#w3
      Contact( "Input".Ss_Low_XiloB2 )
      Contact( "DB_TrungGian".Xung_200ms )
      Add(in1 := "Output".Act_Weight_XiloB2, in2 := "M_Inverter", out => "Output".Act_Weight_XiloB2)
   END_RUNG
   RUNG wire#w1
      { S7_Templates := "SrcType := Real" } GE_Contact(in1 := "Input_Data".Load_ScaleB, in2 := #sum2_Xilo)
      { S7_Templates := "SrcType := Real" } LT_Contact(in1 := "Input_Data".Load_ScaleB, in2 := "Input_Data".Set_Weight_DauKho)
      wire#w4
      Move(in := #sum1_Xilo, out1 => "Output".Act_Weight_XiloB2)
      Coil( "Input".Ss_Low_XiloB3 )
   END_RUNG
   RUNG wire#w4
      Contact( "Input".Ss_Low_XiloB3 )
      Contact( "DB_TrungGian".Xung_200ms )
      Add(in1 := "Output".Act_Weight_XiloB3, in2 := "M_Inverter", out => "Output".Act_Weight_XiloB3)
   END_RUNG
   RUNG wire#w1
      { S7_Templates := "SrcType := Real" } GE_Contact(in1 := "Input_Data".Load_ScaleB, in2 := "Input_Data".Set_Weight_DauKho)
      Move(in := #sum1_Xilo, out1 => "Output".Act_Weight_XiloB3)
   END_RUNG
   // the same network as SCL:
   #_w1 := "M_Auto_Motor_Tai" AND "Input".Ss_ScalesA AND "TimeDelay".Q;
   "Input".Ss_Low_XiloB1 := #_w1 AND ("Input_Data".Load_ScaleB < #sum1_Xilo);
   IF "Input".Ss_Low_XiloB1 AND "Input".Ss_Low_XiloB1 AND "DB_TrungGian".Xung_200ms THEN
       "Output".Act_Weight_XiloB1 := "Output".Act_Weight_XiloB1 + "M_Inverter";
   END_IF;
   #_w2 := #_w1 AND ("Input_Data".Load_ScaleB >= #sum1_Xilo) AND ("Input_Data".Load_ScaleB < #sum2_Xilo);
   IF #_w2 THEN "Output".Act_Weight_XiloB1 := #sum1_Xilo; END_IF;
   "Input".Ss_Low_XiloB2 := #_w2;
   IF #_w2 AND "Input".Ss_Low_XiloB2 AND "DB_TrungGian".Xung_200ms THEN
       "Output".Act_Weight_XiloB2 := "Output".Act_Weight_XiloB2 + "M_Inverter";
   END_IF;
   #_w3 := #_w1 AND ("Input_Data".Load_ScaleB >= #sum2_Xilo) AND ("Input_Data".Load_ScaleB < "Input_Data".Set_Weight_DauKho);
   IF #_w3 THEN "Output".Act_Weight_XiloB2 := #sum1_Xilo; END_IF;
   "Input".Ss_Low_XiloB3 := #_w3;
   IF #_w3 AND "Input".Ss_Low_XiloB3 AND "DB_TrungGian".Xung_200ms THEN
       "Output".Act_Weight_XiloB3 := "Output".Act_Weight_XiloB3 + "M_Inverter";
   END_IF;
   IF #_w1 AND ("Input_Data".Load_ScaleB >= "Input_Data".Set_Weight_DauKho) THEN
       "Output".Act_Weight_XiloB3 := #sum1_Xilo;
   END_IF;
END_REGION

REGION Network 3
   RUNG wire#powerrail
      I_Contact( "M_Auto_Motor_Tai" )
      Contact( "M_Step2" )
      Move(in := 0.0, out1 => "Output".Act_Weight_XiloB1, out2 => "Output".Act_Weight_XiloB2, out3 => "Output".Act_Weight_XiloB3)
   END_RUNG
   // the same network as SCL:
   IF NOT "M_Auto_Motor_Tai" AND "M_Step2" THEN
       "Output".Act_Weight_XiloB1 := 0.0;
       "Output".Act_Weight_XiloB2 := 0.0;
       "Output".Act_Weight_XiloB3 := 0.0;
   END_IF;
END_REGION
END_FUNCTION

FUNCTION "FC_XiloBotCa" : Void   // FC10, LAD
{ S7_Optimized_Access := 'TRUE' }
VERSION : 0.1
   VAR_TEMP
      sum1_Xilo : Real;
      sum2_Xilo : Real;
      sum3_Xilo : Real;
      "1" : Real;
      "2" : Real;
      "3" : Real;
   END_VAR
   VAR_TEMP   // added for the SCL form of the ladder/FBD networks
      _w1 : Bool;
      _w2 : Bool;
      _w3 : Bool;
   END_VAR
BEGIN

REGION Network 1: k.lượng bột cá =e
   // tính các giá trị e/4, 2e/4 , 3e/4, 
   // tính các g.trị d+ e/4 , d+ 2e/4, d+3e/4
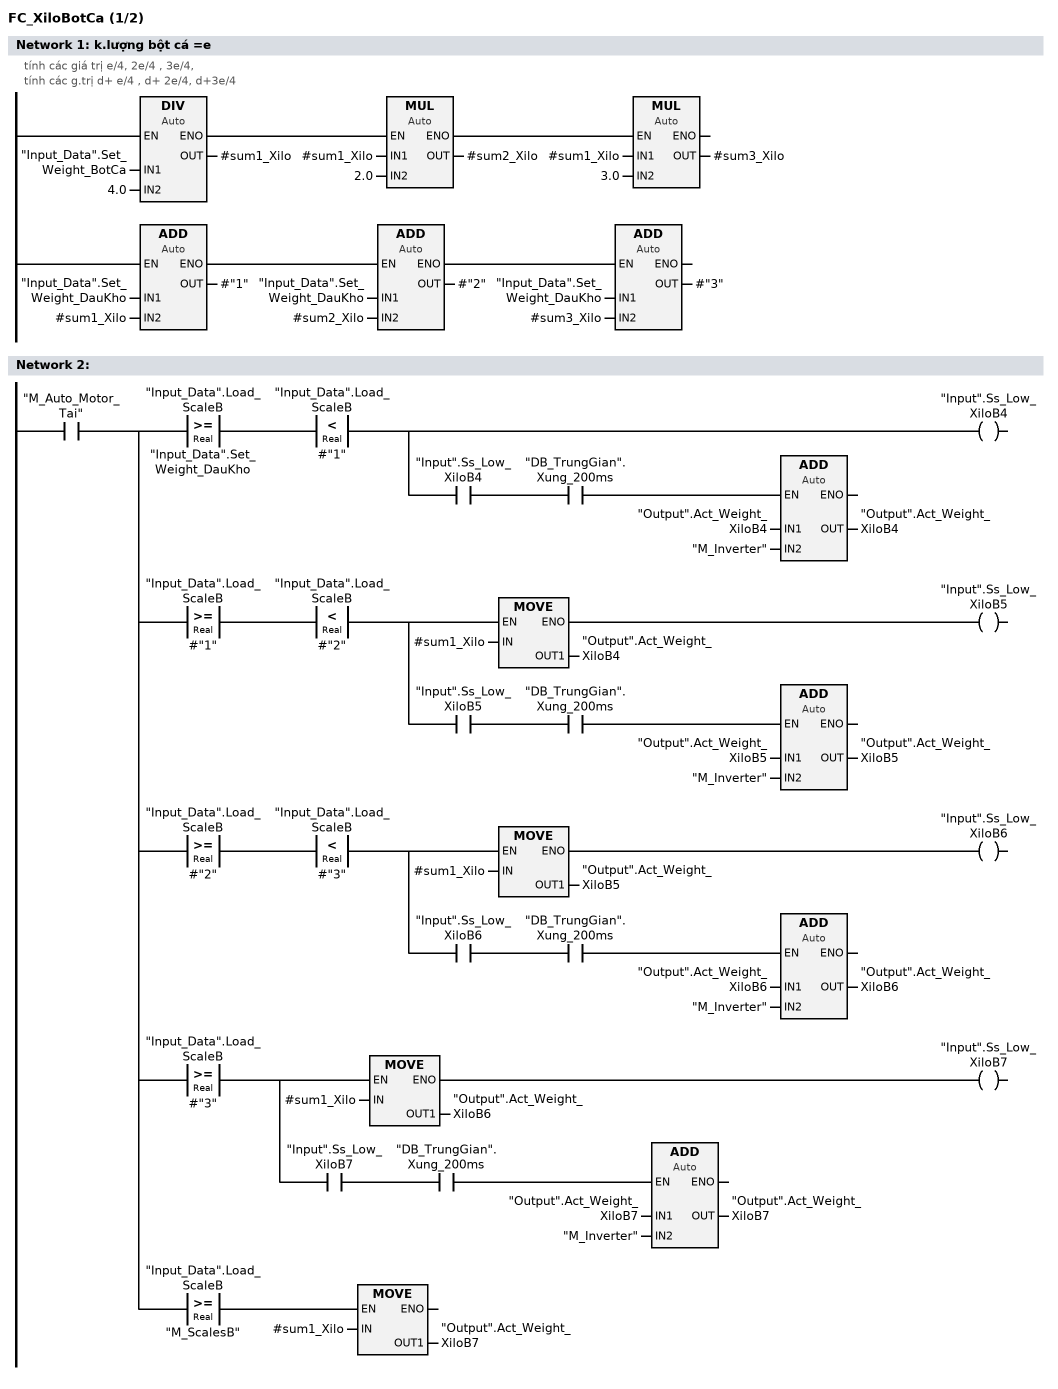
   RUNG wire#powerrail
      Div(in1 := "Input_Data".Set_Weight_BotCa, in2 := 4.0, out => #sum1_Xilo)
      Mul(in1 := #sum1_Xilo, in2 := 2.0, out => #sum2_Xilo)
      Mul(in1 := #sum1_Xilo, in2 := 3.0, out => #sum3_Xilo)
   END_RUNG
   RUNG wire#powerrail
      Add(in1 := "Input_Data".Set_Weight_DauKho, in2 := #sum1_Xilo, out => #"1")
      Add(in1 := "Input_Data".Set_Weight_DauKho, in2 := #sum2_Xilo, out => #"2")
      Add(in1 := "Input_Data".Set_Weight_DauKho, in2 := #sum3_Xilo, out => #"3")
   END_RUNG
   // the same network as SCL:
   #sum1_Xilo := "Input_Data".Set_Weight_BotCa / 4.0;
   #sum2_Xilo := #sum1_Xilo * 2.0;
   #sum3_Xilo := #sum1_Xilo * 3.0;
   #"1" := "Input_Data".Set_Weight_DauKho + #sum1_Xilo;
   #"2" := "Input_Data".Set_Weight_DauKho + #sum2_Xilo;
   #"3" := "Input_Data".Set_Weight_DauKho + #sum3_Xilo;
END_REGION

REGION Network 2
   RUNG wire#powerrail
      Contact( "M_Auto_Motor_Tai" )
      wire#w1
      { S7_Templates := "SrcType := Real" } GE_Contact(in1 := "Input_Data".Load_ScaleB, in2 := "Input_Data".Set_Weight_DauKho)
      { S7_Templates := "SrcType := Real" } LT_Contact(in1 := "Input_Data".Load_ScaleB, in2 := #"1")
      wire#w2
      Coil( "Input".Ss_Low_XiloB4 )
   END_RUNG
   RUNG wire#w2
      Contact( "Input".Ss_Low_XiloB4 )
      Contact( "DB_TrungGian".Xung_200ms )
      Add(in1 := "Output".Act_Weight_XiloB4, in2 := "M_Inverter", out => "Output".Act_Weight_XiloB4)
   END_RUNG
   RUNG wire#w1
      { S7_Templates := "SrcType := Real" } GE_Contact(in1 := "Input_Data".Load_ScaleB, in2 := #"1")
      { S7_Templates := "SrcType := Real" } LT_Contact(in1 := "Input_Data".Load_ScaleB, in2 := #"2")
      wire#w3
      Move(in := #sum1_Xilo, out1 => "Output".Act_Weight_XiloB4)
      Coil( "Input".Ss_Low_XiloB5 )
   END_RUNG
   RUNG wire#w3
      Contact( "Input".Ss_Low_XiloB5 )
      Contact( "DB_TrungGian".Xung_200ms )
      Add(in1 := "Output".Act_Weight_XiloB5, in2 := "M_Inverter", out => "Output".Act_Weight_XiloB5)
   END_RUNG
   RUNG wire#w1
      { S7_Templates := "SrcType := Real" } GE_Contact(in1 := "Input_Data".Load_ScaleB, in2 := #"2")
      { S7_Templates := "SrcType := Real" } LT_Contact(in1 := "Input_Data".Load_ScaleB, in2 := #"3")
      wire#w4
      Move(in := #sum1_Xilo, out1 => "Output".Act_Weight_XiloB5)
      Coil( "Input".Ss_Low_XiloB6 )
   END_RUNG
   RUNG wire#w4
      Contact( "Input".Ss_Low_XiloB6 )
      Contact( "DB_TrungGian".Xung_200ms )
      Add(in1 := "Output".Act_Weight_XiloB6, in2 := "M_Inverter", out => "Output".Act_Weight_XiloB6)
   END_RUNG
   RUNG wire#w1
      { S7_Templates := "SrcType := Real" } GE_Contact(in1 := "Input_Data".Load_ScaleB, in2 := #"3")
      wire#w5
      Move(in := #sum1_Xilo, out1 => "Output".Act_Weight_XiloB6)
      Coil( "Input".Ss_Low_XiloB7 )
   END_RUNG
   RUNG wire#w5
      Contact( "Input".Ss_Low_XiloB7 )
      Contact( "DB_TrungGian".Xung_200ms )
      Add(in1 := "Output".Act_Weight_XiloB7, in2 := "M_Inverter", out => "Output".Act_Weight_XiloB7)
   END_RUNG
   RUNG wire#w1
      { S7_Templates := "SrcType := Real" } GE_Contact(in1 := "Input_Data".Load_ScaleB, in2 := "M_ScalesB")
      Move(in := #sum1_Xilo, out1 => "Output".Act_Weight_XiloB7)
   END_RUNG
   // the same network as SCL:
   "Input".Ss_Low_XiloB4 := "M_Auto_Motor_Tai" AND ("Input_Data".Load_ScaleB >= "Input_Data".Set_Weight_DauKho) AND ("Input_Data".Load_ScaleB < #"1");
   IF "Input".Ss_Low_XiloB4 AND "Input".Ss_Low_XiloB4 AND "DB_TrungGian".Xung_200ms THEN
       "Output".Act_Weight_XiloB4 := "Output".Act_Weight_XiloB4 + "M_Inverter";
   END_IF;
   #_w1 := "M_Auto_Motor_Tai" AND ("Input_Data".Load_ScaleB >= #"1") AND ("Input_Data".Load_ScaleB < #"2");
   IF #_w1 THEN "Output".Act_Weight_XiloB4 := #sum1_Xilo; END_IF;
   "Input".Ss_Low_XiloB5 := #_w1;
   IF #_w1 AND "Input".Ss_Low_XiloB5 AND "DB_TrungGian".Xung_200ms THEN
       "Output".Act_Weight_XiloB5 := "Output".Act_Weight_XiloB5 + "M_Inverter";
   END_IF;
   #_w2 := "M_Auto_Motor_Tai" AND ("Input_Data".Load_ScaleB >= #"2") AND ("Input_Data".Load_ScaleB < #"3");
   IF #_w2 THEN "Output".Act_Weight_XiloB5 := #sum1_Xilo; END_IF;
   "Input".Ss_Low_XiloB6 := #_w2;
   IF #_w2 AND "Input".Ss_Low_XiloB6 AND "DB_TrungGian".Xung_200ms THEN
       "Output".Act_Weight_XiloB6 := "Output".Act_Weight_XiloB6 + "M_Inverter";
   END_IF;
   #_w3 := "M_Auto_Motor_Tai" AND ("Input_Data".Load_ScaleB >= #"3");
   IF #_w3 THEN "Output".Act_Weight_XiloB6 := #sum1_Xilo; END_IF;
   "Input".Ss_Low_XiloB7 := #_w3;
   IF #_w3 AND "Input".Ss_Low_XiloB7 AND "DB_TrungGian".Xung_200ms THEN
       "Output".Act_Weight_XiloB7 := "Output".Act_Weight_XiloB7 + "M_Inverter";
   END_IF;
   IF "M_Auto_Motor_Tai" AND ("Input_Data".Load_ScaleB >= "M_ScalesB") THEN
       "Output".Act_Weight_XiloB7 := #sum1_Xilo;
   END_IF;
END_REGION

REGION Network 3
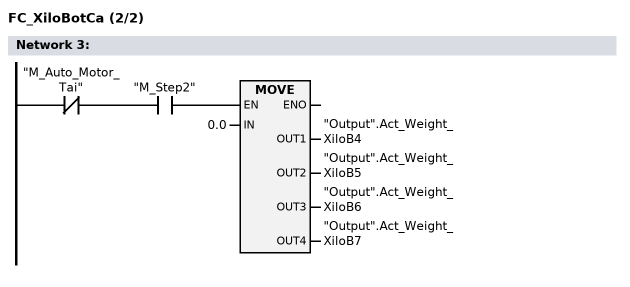
   RUNG wire#powerrail
      I_Contact( "M_Auto_Motor_Tai" )
      Contact( "M_Step2" )
      Move(in := 0.0, out1 => "Output".Act_Weight_XiloB4, out2 => "Output".Act_Weight_XiloB5, out3 => "Output".Act_Weight_XiloB6, out4 => "Output".Act_Weight_XiloB7)
   END_RUNG
   // the same network as SCL:
   IF NOT "M_Auto_Motor_Tai" AND "M_Step2" THEN
       "Output".Act_Weight_XiloB4 := 0.0;
       "Output".Act_Weight_XiloB5 := 0.0;
       "Output".Act_Weight_XiloB6 := 0.0;
       "Output".Act_Weight_XiloB7 := 0.0;
   END_IF;
END_REGION
END_FUNCTION

ORGANIZATION_BLOCK "Main"   // OB1, LAD, ProgramCycle
TITLE = "Main Program Sweep (Cycle)"
{ S7_Optimized_Access := 'TRUE' }
VERSION : 0.1
   VAR_INPUT
      Initial_Call : Bool;   // Initial call of this OB
      Remanence : Bool;   // =True, if remanent data are available
   END_VAR
   VAR_TEMP   // added for the SCL form of the ladder/FBD networks
      _w1 : Bool;
   END_VAR
BEGIN

REGION Network 1: chọn chế độ vận hành
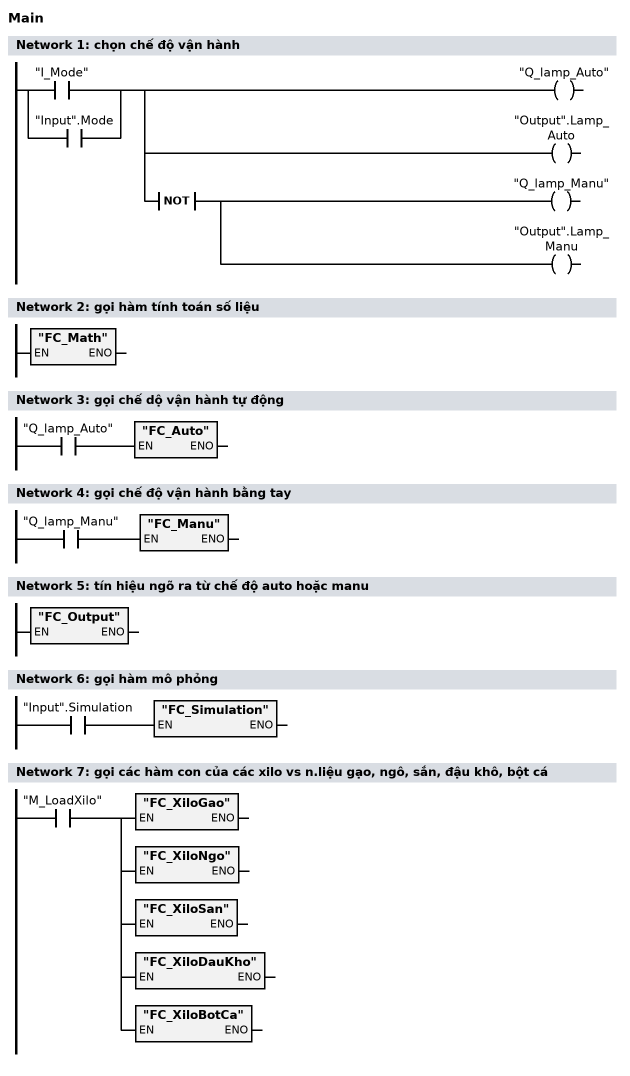
   RUNG wire#powerrail
      Contact( "I_Mode" )
      wire#w1
      Coil( "Q_lamp_Auto" )
   END_RUNG
   RUNG wire#powerrail
      Contact( "Input".Mode )
   END_RUNG wire#w1
   RUNG wire#w1
      Coil( "Output".Lamp_Auto )
   END_RUNG
   RUNG wire#w1
      Not()
      wire#w2
      Coil( "Q_lamp_Manu" )
   END_RUNG
   RUNG wire#w2
      Coil( "Output".Lamp_Manu )
   END_RUNG
   // the same network as SCL:
   "Q_lamp_Auto" := "I_Mode" OR "Input".Mode;
   "Output".Lamp_Auto := "Q_lamp_Auto";
   "Q_lamp_Manu" := NOT "Q_lamp_Auto";
   "Output".Lamp_Manu := NOT "Q_lamp_Auto";
END_REGION

REGION Network 2: gọi hàm tính toán số liệu
   RUNG wire#powerrail
      "FC_Math"()
   END_RUNG
   // the same network as SCL:
   "FC_Math"();
END_REGION

REGION Network 3: gọi chế dộ vận hành tự động
   RUNG wire#powerrail
      Contact( "Q_lamp_Auto" )
      "FC_Auto"()
   END_RUNG
   // the same network as SCL:
   IF "Q_lamp_Auto" THEN "FC_Auto"(); END_IF;
END_REGION

REGION Network 4: gọi chế độ vận hành bằng tay
   RUNG wire#powerrail
      Contact( "Q_lamp_Manu" )
      "FC_Manu"()
   END_RUNG
   // the same network as SCL:
   IF "Q_lamp_Manu" THEN "FC_Manu"(); END_IF;
END_REGION

REGION Network 5: tín hiệu ngõ ra từ chế độ auto hoặc manu
   RUNG wire#powerrail
      "FC_Output"()
   END_RUNG
   // the same network as SCL:
   "FC_Output"();
END_REGION

REGION Network 6: gọi hàm mô phỏng
   RUNG wire#powerrail
      Contact( "Input".Simulation )
      "FC_Simulation"()
   END_RUNG
   // the same network as SCL:
   IF "Input".Simulation THEN "FC_Simulation"(); END_IF;
END_REGION

REGION Network 7: gọi các hàm con của các xilo vs n.liệu gạo, ngô, sắn, đậu khô, bột cá
   RUNG wire#powerrail
      Contact( "M_LoadXilo" )
      wire#w1
      "FC_XiloGao"()
   END_RUNG
   RUNG wire#w1
      "FC_XiloNgo"()
   END_RUNG
   RUNG wire#w1
      "FC_XiloSan"()
   END_RUNG
   RUNG wire#w1
      "FC_XiloDauKho"()
   END_RUNG
   RUNG wire#w1
      "FC_XiloBotCa"()
   END_RUNG
   // the same network as SCL:
   #_w1 := "M_LoadXilo";
   IF #_w1 THEN
       "FC_XiloGao"();
       "FC_XiloNgo"();
       "FC_XiloSan"();
       "FC_XiloDauKho"();
       "FC_XiloBotCa"();
   END_IF;
END_REGION
END_ORGANIZATION_BLOCK